PROPERTY ModuleSide : Tc3_Xts_Utility.ModuleSide
GET
ModuleSide := _ModuleSide;
END_GET
SET
_ModuleSide := ModuleSide;
END_SET
END_PROPERTY

PROPERTY Offset : ST_OriginTransform
GET
Offset := _Offset;
END_GET
SET
_Offset := Offset;
END_SET
END_PROPERTY

PROPERTY OTCID : OTCID
GET
OTCID := _Otcid;
END_GET
SET
_Otcid := OTCID;
END_SET
END_PROPERTY

END_FUNCTION_BLOCK

// _Internal/Parts/Tasks/InitializeXtsPartTask
{attribute 'no_explicit_call' := 'This FB is a CLASS and must be accessed using methods or properties'}
FUNCTION_BLOCK InitializeXtsPartTask EXTENDS BaseTaskResult IMPLEMENTS I_XtsPartInitializeTask
VAR
	_Initialized : BOOL;
	_PartId		 : I_XtsPartId;
	_PartUtility : I_ContainXtsPartUtility;
	_Parent		 : I_ContainComponents;
	_Properties	 : I_ContainXtsPartProperties;

	//
	_XtsModuleCollection : I_ContainXtsModules;

	//
	_SubState : UDINT;
END_VAR

METHOD Initialize
VAR
	Module : I_XtsModule;
	pModule	 : POINTER TO XtsModule;
END_VAR
CASE _SubState OF
	0:
		IF _Initialized THEN
			RETURN;
		END_IF

		_Busy	  := TRUE;
		_Error	  := FALSE;
		_ErrorId  := 0;
		_SubState := 10;

	10:
		IF _PartUtility.Utility.GetModuleOids() THEN
			IF _PartUtility.Utility.P_ModuleCount < 1 THEN
				_SubState := 100;
			END_IF

			_XtsModuleCollection.XtsModules.Create(UDINT_TO_UINT(_PartUtility.Utility.P_ModuleCount));
			_SubState := 20;
		END_IF

	20:
		_XtsModuleCollection.XtsModules.ResetIterator();
		WHILE _XtsModuleCollection.XtsModules.MoveToNext DO
			Module := _XtsModuleCollection.XtsModules.Current;
			Module.RegisterWithParent(_Parent);
			Module.Id	   := _XtsModuleCollection.XtsModules.CurrentItem;
			Module.Otcid   := _PartUtility.Utility.P_ModuleOids[_XtsModuleCollection.XtsModules.CurrentItem];
			Module.Utility := _PartUtility.Utility.ModuleTcIo(UDINT_TO_UINT(_XtsModuleCollection.XtsModules.CurrentItem));
		END_WHILE

		_SubState := 30;

	30:
		_Properties.Properties.General.ModuleSide := _PartUtility.Utility.GetModuleSide();
		_Properties.Properties.General.Offset	  := _PartUtility.Utility.GetOriginTransform();
		_Properties.Properties.General.OTCID	  := _PartUtility.Utility.GetTaskOid();
		_SubState								  := 100;

	100:
		_Initialized := TRUE;
		_Busy		 := FALSE;
		_SubState	 := 0;
END_CASE
END_METHOD

{attribute 'monitoring':='call'}
PROPERTY Initialized : BOOL
GET
Initialized := _Initialized;
END_GET
SET
_Initialized := Initialized;
END_SET
END_PROPERTY

PROPERTY XtsPartId : I_XtsPartId
GET
END_GET
SET
_PartId := XtsPartId;
__QUERYINTERFACE(_PartId, _PartUtility);
__QUERYINTERFACE(_PartId, _XtsModuleCollection);
__QUERYINTERFACE(_PartId, _Parent);
__QUERYINTERFACE(_PartId, _Properties);
END_SET
END_PROPERTY

END_FUNCTION_BLOCK

// _Internal/TaskBase/BaseTaskResult
{attribute 'hide_all_locals'}
FUNCTION_BLOCK BaseTaskResult IMPLEMENTS I_TaskResult
VAR
	_TaskName : T_MaxString;
	_Busy	 : BOOL;
	_Error	 : BOOL;
	_ErrorId : UDINT;
END_VAR

{attribute 'monitoring' := 'call'}
PROPERTY Busy : BOOL
GET
Busy := _Busy;
END_GET
END_PROPERTY

{attribute 'monitoring' := 'call'}
PROPERTY Error : BOOL
GET
Error := _Error;
END_GET
END_PROPERTY

{attribute 'monitoring' := 'call'}
PROPERTY ErrorId : UDINT
GET
ErrorId := _ErrorId;
END_GET
END_PROPERTY

{attribute 'monitoring':='call'}
PROPERTY TaskName : STRING
GET
TaskName := _TaskName;
END_GET
SET
_TaskName := TaskName;
END_SET
END_PROPERTY

END_FUNCTION_BLOCK

// _Internal/Parts/Tasks/Interfaces/I_XtsPartInitializeTask
INTERFACE I_XtsPartInitializeTask EXTENDS I_XtsPartTask, I_Initializable

END_INTERFACE

// _Internal/Parts/Tasks/Interfaces/I_XtsPartTask
INTERFACE I_XtsPartTask EXTENDS I_XtsPartTaskResult

PROPERTY XtsPartId : I_XtsPartId
GET
END_GET
SET
END_SET
END_PROPERTY

END_INTERFACE

// _Internal/Parts/Tasks/Interfaces/I_XtsPartTaskResult
INTERFACE I_XtsPartTaskResult EXTENDS I_TaskResult

END_INTERFACE

// _Internal/Collections/Modules/ModuleCollection/XtsModuleCollection
{attribute 'no_explicit_call' := 'This FB is a CLASS and must be accessed using methods or properties'}
{attribute 'enable_dynamic_creation'}
FUNCTION_BLOCK XtsModuleCollection IMPLEMENTS I_XtsModuleCollection, I_Peekable
VAR
	pModuleBuffer	 : POINTER TO PVOID;
	_NumberOfModules : UINT;
	_CurrentModule : I_XtsModule;
	_CurrentIndex  : UDINT := 0;
	{attribute 'hide'}
	_CollectionAdapter : XtsModuleCollectionAdapter(THIS^);
END_VAR

METHOD Clear
VAR
	i	   : UDINT;
	Module : POINTER TO XtsModule;
END_VAR
IF IsEmpty THEN
	RETURN;
END_IF

FOR i := 1 TO _NumberOfModules DO
	Module := GetModuleInstance(i);
	IF Module <> ADR(NullObjects.XtsModule) THEN
		__DELETE(Module);
	END_IF
END_FOR

__DELETE(pModuleBuffer);
_NumberOfModules := 0;
END_METHOD

{attribute 'monitoring' := 'call'}
PROPERTY Count : UDINT
GET
Count := _NumberOfModules;
END_GET
END_PROPERTY

{attribute 'hide'}
METHOD Create : BOOL
VAR_INPUT
	NumberOfModules : UINT;
END_VAR

VAR
	i		 : UINT;
	pModule	 : POINTER TO XtsModule;
	ppBuffer : POINTER TO POINTER TO XtsModule;
END_VAR
IF NOT IsEmpty THEN
	Clear();
END_IF

_NumberOfModules := NumberOfModules;
pModuleBuffer	 := __NEW(PVOID, NumberOfModules);
IF pModuleBuffer <> 0 THEN
	FOR i := 1 TO _NumberOfModules DO
		pModule	  := __NEW(XtsModule(Name := CONCAT('Module ',UINT_TO_STRING(i))));
		ppBuffer  := pModuleBuffer + ((i - 1) * SIZEOF(PVOID));
		ppBuffer^ := pModule;
	END_FOR

	Create := TRUE;
END_IF
END_METHOD

METHOD GetById : I_XtsModule
VAR_INPUT
	ModuleId	: UDINT;
END_VAR
GetById := GetModuleInstance(ModuleId)^;
END_METHOD

METHOD GetByOtcid : I_XtsModule
VAR_INPUT
	ModuleOtcid	: OTCID;
END_VAR
VAR
	i : UDINT;
	ppModule : POINTER TO POINTER TO XtsModule;
END_VAR
GetByOtcid := NullObjects.XtsModule;
FOR i := 0 TO _NumberOfModules DO
	ppModule := pModuleBuffer + ((i) * SIZEOF(PVOID));
	IF ppModule^^.Otcid = ModuleOtcid THEN
		GetByOtcid := ppModule^^;
		RETURN;
	END_IF
END_FOR
END_METHOD

{attribute 'monitoring' := 'call'}
PROPERTY IsEmpty : BOOL
GET
IsEmpty := _NumberOfModules = 0;
END_GET
END_PROPERTY

{attribute 'monitoring':='call'}
PROPERTY Current : I_XtsModule
GET
IF _CurrentModule = 0 THEN
	Current := NullObjects.XtsModule;
ELSE
	Current := _CurrentModule;
END_IF
END_GET
END_PROPERTY

{attribute 'monitoring' := 'call'}
PROPERTY CurrentItem : UDINT
GET
CurrentItem := _CurrentIndex;
END_GET
END_PROPERTY

PROPERTY MoveToNext : BOOL
GET
MoveToNext := FALSE;
IF _NumberOfModules = 0 THEN
	RETURN;
END_IF

IF _CurrentIndex = _NumberOfModules THEN
	RETURN;
END_IF

_CurrentModule := GetById(_CurrentIndex + 1);
_CurrentIndex  := _CurrentIndex + 1;
MoveToNext	   := TRUE;
END_GET
END_PROPERTY

METHOD ResetIterator
_CurrentModule := NullObjects.XtsModule;
_CurrentIndex  := 0;
END_METHOD

METHOD Dispose
VAR
	pDispose : POINTER TO XtsModuleCollection;
END_VAR
Clear();
pDispose := THIS;
__DELETE(pDispose);
END_METHOD

//FB_Exit must be implemented explicitly. If there is an implementation, then the
//method is called before the controller removes the code of the function block instance
//(implicit call). The return value is not evaluated.
METHOD FB_Exit: BOOL
VAR_INPUT
    bInCopyCode: BOOL;  // TRUE: the exit method is called in order to leave the instance which will be copied afterwards (online change).  
END_VAR
IF bInCopyCode THEN
	RETURN;
END_IF

Clear();
END_METHOD

METHOD AcceptPeeker
VAR_INPUT
	Peeker	: Core.I_Peeker;
END_VAR
Peeker.PeekCollection(_CollectionAdapter);
END_METHOD

METHOD PROTECTED CheckModuleId : BOOL
VAR_INPUT
	ModuleId : UDINT;
END_VAR
CheckModuleId := (ModuleId > 0) AND (ModuleId <= _NumberOfModules) AND (pModuleBuffer <> 0);
END_METHOD

METHOD PROTECTED GetModuleInstance : POINTER TO XtsModule
VAR_INPUT
	ModuleId : UDINT; // 1 based index
END_VAR

VAR
	ppModule : POINTER TO POINTER TO XtsModule;
END_VAR
IF CheckModuleId(ModuleId) THEN
	ppModule := pModuleBuffer + ((ModuleId - 1) * SIZEOF(PVOID));
	GetModuleInstance := ppModule^;
ELSE
	GetModuleInstance := ADR(NullObjects.XtsModule);
END_IF
END_METHOD

END_FUNCTION_BLOCK

// _Internal/Collections/Modules/ModuleCollection/Interfaces/XtsModuleCollectionAdapter
FUNCTION_BLOCK XtsModuleCollectionAdapter IMPLEMENTS I_Collection
VAR
	_ModuleCollection : I_XtsModuleCollection;
END_VAR

METHOD AddItem
VAR_INPUT
	Item	: Core.I_Base;
END_VAR
END_METHOD

METHOD Clear
_ModuleCollection.Clear();
END_METHOD

{attribute 'monitoring' := 'call'}
PROPERTY Count : UDINT
GET
Count := _ModuleCollection.Count;
END_GET
END_PROPERTY

PROPERTY Current : Core.I_Base
GET
Current := _ModuleCollection.Current;
END_GET
END_PROPERTY

{attribute 'monitoring' := 'call'}
PROPERTY CurrentItem : UDINT
GET
CurrentItem := _ModuleCollection.CurrentItem;
END_GET
END_PROPERTY

//FB_Init is always available implicitly and it is used primarily for initialization.
//The return value is not evaluated. For a specific influence, you can also declare the
//methods explicitly and provide additional code there with the standard initialization
//code. You can evaluate the return value.
METHOD FB_Init: BOOL
VAR_INPUT
    bInitRetains: BOOL; // TRUE: the retain variables are initialized (reset warm / reset cold)
    bInCopyCode: BOOL;  // TRUE: the instance will be copied to the copy code afterward (online change)
	XtsModuleCollection : I_XtsModuleCollection;   
END_VAR
_ModuleCollection := XtsModuleCollection;
END_METHOD

{attribute 'monitoring' := 'call'}
PROPERTY IsEmpty : BOOL
GET
IsEmpty := _ModuleCollection.IsEmpty;
END_GET
END_PROPERTY

PROPERTY MoveToNext : BOOL
GET
MoveToNext := _ModuleCollection.MoveToNext;
END_GET
END_PROPERTY

METHOD RemoveItem
VAR_INPUT
	Item	: Core.I_Base;
END_VAR
END_METHOD

METHOD ResetIterator
_ModuleCollection.ResetIterator();
END_METHOD

END_FUNCTION_BLOCK

// _Internal/XtsSystem/Properties/Interfaces/I_ContainXtsSystemProperties
INTERFACE I_ContainXtsSystemProperties EXTENDS I_Base

PROPERTY UtilityProperties : I_XtsSystemUtilityProperties
GET
END_GET
END_PROPERTY

END_INTERFACE

// _Internal/XtsSystem/Properties/Interfaces/I_XtsSystemUtilityProperties
INTERFACE I_XtsSystemUtilityProperties EXTENDS I_Base

PROPERTY Mover : I_XtsSystemUtilityPropertiesMover
GET
END_GET
END_PROPERTY

END_INTERFACE

// _Internal/XtsSystem/Properties/Interfaces/I_XtsSystemUtilityPropertiesMover
INTERFACE I_XtsSystemUtilityPropertiesMover EXTENDS I_Base

PROPERTY XtsMagnetPlateType : MagnetPlateType
GET
END_GET
SET
END_SET
END_PROPERTY

PROPERTY XtsMoverType : MoverType
GET
END_GET
SET
END_SET
END_PROPERTY

END_INTERFACE

// _Internal/XtsSystem/Status/Interfaces/I_ContainXtsSystemStatus
INTERFACE I_ContainXtsSystemStatus EXTENDS I_Base

{attribute 'monitoring':='call'}
PROPERTY Status : I_XtsSystemStatus
GET
END_GET
END_PROPERTY

END_INTERFACE

// _Internal/XtsSystem/Status/Interfaces/I_XtsSystemStatus
INTERFACE I_XtsSystemStatus EXTENDS I_Base, I_Cyclic

{attribute 'monitoring':='call'}
PROPERTY NumberOfMovers : UDINT
GET
END_GET
END_PROPERTY

{attribute 'monitoring':='call'}
PROPERTY NumberOfParts : UDINT
GET
END_GET
END_PROPERTY

{attribute 'monitoring':='call'}
PROPERTY NumberOfPositionTriggers : UDINT
GET
END_GET
END_PROPERTY

{attribute 'monitoring':='call'}
PROPERTY NumberOfStations : UDINT
GET
END_GET
END_PROPERTY

{attribute 'monitoring':='call'}
PROPERTY NumberOfTracks : UDINT
GET
END_GET
END_PROPERTY

{attribute 'monitoring':='call'}
PROPERTY NumberOfZones : UDINT
GET
END_GET
END_PROPERTY

{attribute 'monitoring':='call'}
PROPERTY NumberPartsNotReady : USINT
GET
END_GET
END_PROPERTY

{attribute 'monitoring':='call'}
PROPERTY NumberPartsReady : USINT
GET
END_GET
END_PROPERTY

{attribute 'monitoring':='call'}
PROPERTY Simulated : BOOL
GET
END_GET
END_PROPERTY

{attribute 'monitoring':='call'}
PROPERTY Vdc24Okay : BOOL
GET
END_GET
END_PROPERTY

{attribute 'monitoring':='call'}
PROPERTY Vdc48Okay : BOOL
GET
END_GET
END_PROPERTY

END_INTERFACE

// XtsSystem/Interfaces/I_XtsSystemConfiguration
INTERFACE I_XtsSystemConfiguration EXTENDS I_Base

{attribute 'monitoring':='call'}
PROPERTY CommandPositionTriggersOnDisable : BOOL
GET
END_GET
SET
END_SET
END_PROPERTY

{attribute 'monitoring':='call'}
PROPERTY CommandPositionTriggersOnEnable : BOOL
GET
END_GET
SET
END_SET
END_PROPERTY

{attribute 'monitoring':='call'}
PROPERTY CommandStationsOnDisable : BOOL
GET
END_GET
SET
END_SET
END_PROPERTY

{attribute 'monitoring':='call'}
PROPERTY CommandStationsOnEnable : BOOL
GET
END_GET
SET
END_SET
END_PROPERTY

END_INTERFACE

// _Internal/XtsSystem/Base/Interfaces/I_XtsTask
INTERFACE I_XtsTask EXTENDS I_XtsTaskResult

{attribute 'monitoring' := 'call'}
PROPERTY XpuId : I_XtsXpuId
GET
END_GET
SET
END_SET
END_PROPERTY

END_INTERFACE

// _Internal/XtsSystem/Base/Interfaces/I_XtsTaskResult
INTERFACE I_XtsTaskResult EXTENDS I_TaskResult

{attribute 'monitoring':='call'}
PROPERTY TaskId : XtsSystemTaskId
GET
END_GET
END_PROPERTY

END_INTERFACE

// _Internal/XtsSystem/ManualDebugger
FUNCTION_BLOCK ManualDebugger
VAR
	//Xts System Movers Collection
	Movers : CollectionPeeker<5>;
	//Xts System Stations Collection
	Stations : CollectionPeeker<5>;
	//Xts System PositionTriggers Collection
	PositionTriggers : CollectionPeeker<5>;
	//Xts System Zones Collection
	Zones : CollectionPeeker<5>;
	//Xts System XtsParts Collection
	Parts : CollectionPeeker<5>;
	{attribute 'hide'}
	_PartCollection : I_XtsPartCollection;
	//Part defined by PartIdForModules XtsModule Collection
	Modules : CollectionPeeker<5>;
	{attribute 'hide'}
	_PartId			: UDINT := 1;
END_VAR

{attribute 'monitoring':='call'}
PROPERTY PartIdForModules : UDINT
GET
PartIdForModules := _PartId;
END_GET
SET
VAR
	ModulePeekable : I_Peekable;
END_VAR
_PartId := PartIdForModules;

IF __QUERYINTERFACE(_PartCollection.GetById(_PartId).XtsModules, ModulePeekable) THEN
	Modules.CollectionName := CONCAT('Part ', CONCAT(TO_STRING(_PartId), ' Modules'));
	Modules.PeekAt(ModulePeekable);
END_IF
END_SET
END_PROPERTY

PROPERTY RefreshCollections : BOOL
SET
IF NOT RefreshCollections THEN
	RETURN;
END_IF

Movers.Refresh			  := TRUE;
Stations.Refresh		  := TRUE;
PositionTriggers.Refresh := TRUE;
Zones.Refresh			  := TRUE;
Parts.Refresh			  := TRUE;
Modules.Refresh		  := TRUE;
END_SET
END_PROPERTY

METHOD SetCollections
VAR_INPUT
	Movers			 : I_XtsMoverCollection;
	PositionTriggers : I_XtsPositionTriggerCollection;
	Stations		 : I_XtsStationCollection;
	Zones			 : I_XtsZoneCollection;
	Parts			 : I_XtsPartCollection;
END_VAR

VAR
	MoverPeekable	   : I_Peekable;
	PosTriggerPeekable : I_Peekable;
	StationPeekable	   : I_Peekable;
	ZonePeekable	   : I_Peekable;
	PartPeekable	   : I_Peekable;
	ModulePeekable	   : I_Peekable;
END_VAR
IF __QUERYINTERFACE(Movers, MoverPeekable) THEN
	THIS^.Movers.CollectionName := 'Xts System Movers';
	THIS^.Movers.PeekAt(MoverPeekable);
END_IF

IF __QUERYINTERFACE(PositionTriggers, PosTriggerPeekable) THEN
	THIS^.PositionTriggers.CollectionName := 'Xts System Position Triggers';
	THIS^.PositionTriggers.PeekAt(PosTriggerPeekable);
END_IF

IF __QUERYINTERFACE(Stations, StationPeekable) THEN
	THIS^.Stations.CollectionName := 'Xts System Stations';
	THIS^.Stations.PeekAt(StationPeekable);
END_IF

IF __QUERYINTERFACE(Zones, ZonePeekable) THEN
	THIS^.Zones.CollectionName := 'Xts System Zones';
	THIS^.Zones.PeekAt(ZonePeekable);
END_IF

IF __QUERYINTERFACE(Parts, PartPeekable) THEN
	_PartCollection		  := Parts;
	THIS^.Parts.CollectionName := 'Xts System Parts';
	THIS^.Parts.PeekAt(PartPeekable);
END_IF

// IF __QUERYINTERFACE(_PartCollection.GetById(_PartId).XtsModules, ModulePeekable) THEN
// 	THIS^.Modules.CollectionName := CONCAT('Part ', CONCAT(TO_STRING(_PartId), ' Modules'));
// 	THIS^.Modules.PeekAt(ModulePeekable);
// END_IF
END_METHOD

END_FUNCTION_BLOCK

// _Internal/XtsSystem/Base/Interfaces/I_XtsTaskCollection
INTERFACE I_XtsTaskCollection EXTENDS I_Base, I_Cyclic

METHOD AddTask : BOOL
VAR_INPUT
	Task : I_XtsTask;
END_VAR
END_METHOD

METHOD GetTaskById : I_XtsTask
VAR_INPUT
	TaskId : XtsSystemTaskId;
END_VAR
END_METHOD

METHOD GetTaskByName : I_XtsTask
VAR_INPUT
	Name : T_MaxString;
END_VAR
END_METHOD

METHOD RemoveTaskById
VAR_INPUT
	TaskId : XtsSystemTaskId;
END_VAR
END_METHOD

METHOD RemoveTaskByInstance
VAR_INPUT
	Task : I_XtsTask;
END_VAR
END_METHOD

END_INTERFACE

// _Internal/Collections/Movers/MoverCollection/XtsMoverCollection
{attribute 'no_explicit_call' := 'This FB is a CLASS and must be accessed using methods or properties'}
FUNCTION_BLOCK XtsMoverCollection IMPLEMENTS I_XtsMoverCollection, I_Peekable
VAR
	_Collection : Collection<XtsCoreParameters.MaxNumberOfMovers>;
END_VAR

{attribute 'monitoring':='call'}
PROPERTY Current : I_XtsMover
GET
VAR
	Mover : I_XtsMover;
END_VAR
__QUERYINTERFACE(_Collection.Current,Mover);
Current := Mover;
END_GET
END_PROPERTY

{attribute 'monitoring' := 'call'}
PROPERTY CurrentItem : UDINT
GET
CurrentItem := _Collection.CurrentItem;
END_GET
END_PROPERTY

PROPERTY MoveToNext : BOOL
GET
MoveToNext := _Collection.MoveToNext;
END_GET
END_PROPERTY

METHOD ResetIterator
_Collection.ResetIterator();
END_METHOD

METHOD AcceptMoverVisitor
VAR_INPUT
	MoverVisitor : I_XtsMoverVisitor;
END_VAR
VAR
	Mover : I_XtsMover;
END_VAR
_Collection.ResetIterator();
WHILE _Collection.MoveToNext DO
	__QUERYINTERFACE(_Collection.Current, Mover);
	Mover.AcceptMoverVisitor(MoverVisitor);
END_WHILE
END_METHOD

METHOD AcceptPeeker
VAR_INPUT
	Peeker	: Core.I_Peeker;
END_VAR
Peeker.PeekCollection(_Collection);
END_METHOD

METHOD AddItem
VAR_INPUT
	Mover : I_XtsMover;
END_VAR
_Collection.AddItem(Mover);
END_METHOD

METHOD Clear
VAR_INPUT
END_VAR
_Collection.Clear();
END_METHOD

{attribute 'monitoring' := 'call'}
PROPERTY Count : UDINT
GET
Count := _Collection.Count;
END_GET
END_PROPERTY

{attribute 'monitoring':='call'}
PROPERTY IsEmpty : BOOL
GET
IsEmpty := _Collection.IsEmpty;
END_GET
END_PROPERTY

METHOD Map
VAR_INPUT
	Validator : I_XtsMoverValidator;
	Visitor	  : I_XtsMoverVisitor;
END_VAR
VAR
	Mover : I_XtsMover;
END_VAR
_Collection.ResetIterator();
WHILE _Collection.MoveToNext DO
	__QUERYINTERFACE(_Collection.Current, Mover);
	IF Validator.Valid(Mover) THEN
		Visitor.VisitMover(Mover);
	END_IF
END_WHILE
END_METHOD

METHOD Remove
VAR_INPUT
	Mover : I_XtsMover;
END_VAR
_Collection.RemoveItem(Mover);
END_METHOD

END_FUNCTION_BLOCK

// _Internal/Collections/Stations/StationCollection/XtsStationCollection
{attribute 'no_explicit_call' := 'This FB is a CLASS and must be accessed using methods or properties'}
FUNCTION_BLOCK XtsStationCollection IMPLEMENTS I_XtsStationCollection, I_Peekable
VAR
	_Stations : Collection<XtsCoreParameters.MaxNumberOfStations>;
END_VAR

{attribute 'monitoring':='call'}
PROPERTY Current : I_XtsStation
GET
VAR
	Station : I_XtsStation;
END_VAR
__QUERYINTERFACE(_Stations.Current,Station);
Current := Station;
END_GET
END_PROPERTY

{attribute 'monitoring' := 'call'}
PROPERTY CurrentItem : UDINT
GET
CurrentItem := _Stations.CurrentItem;
END_GET
END_PROPERTY

PROPERTY MoveToNext : BOOL
GET
MoveToNext := _Stations.MoveToNext;
END_GET
END_PROPERTY

METHOD ResetIterator
_Stations.ResetIterator();
END_METHOD

METHOD AcceptPeeker
VAR_INPUT
	Peeker	: Core.I_Peeker;
END_VAR
Peeker.PeekCollection(_Stations);
END_METHOD

METHOD AcceptStationVisitor
VAR_INPUT
	StationVisitor : I_XtsStationVisitor;
END_VAR

VAR
	_Station : I_XtsStation;
END_VAR
_Stations.ResetIterator();
WHILE _Stations.MoveToNext DO
	__QUERYINTERFACE(_Stations.Current, _Station);
	_Station.AcceptStationVisitor(StationVisitor);
END_WHILE
END_METHOD

METHOD AddItem
VAR_INPUT
	Station : I_XtsStation;
END_VAR
_Stations.AddItem(Station);
END_METHOD

METHOD Clear
VAR_INPUT
END_VAR
_Stations.Clear();
END_METHOD

{attribute 'monitoring' := 'call'}
PROPERTY Count : UDINT
GET
Count := _Stations.Count;
END_GET
END_PROPERTY

{attribute 'monitoring':='call'}
PROPERTY IsEmpty : BOOL
GET
IsEmpty := _Stations.IsEmpty;
END_GET
END_PROPERTY

METHOD Remove
VAR_INPUT
	Station : I_XtsStation;
END_VAR
_Stations.RemoveItem(Station);
END_METHOD

END_FUNCTION_BLOCK

// _Internal/Collections/PositionTriggers/PositionTriggerCollection/XtsPositionTriggerCollection
{attribute 'no_explicit_call' := 'This FB is a CLASS and must be accessed using methods or properties'}
FUNCTION_BLOCK XtsPositionTriggerCollection IMPLEMENTS I_XtsPositionTriggerCollection, I_Peekable
VAR
	_Collection : Collection<XtsCoreParameters.MaxNumberOfPositionTriggers>;
END_VAR

{attribute 'monitoring':='call'}
PROPERTY Current : I_XtsPositionTrigger
GET
__QUERYINTERFACE(_Collection.Current,Current);
END_GET
END_PROPERTY

{attribute 'monitoring' := 'call'}
PROPERTY CurrentItem : UDINT
GET
CurrentItem := _Collection.CurrentItem;
END_GET
END_PROPERTY

PROPERTY MoveToNext : BOOL
GET
MoveToNext := _Collection.MoveToNext;
END_GET
END_PROPERTY

METHOD ResetIterator
_Collection.ResetIterator();
END_METHOD

METHOD AcceptPeeker
VAR_INPUT
	Peeker	: Core.I_Peeker;
END_VAR
Peeker.PeekCollection(_Collection);
END_METHOD

METHOD AcceptXtsPositionTriggerVisitor
VAR_INPUT
	PositionTriggerVisitor : I_VisitXtsPositionTrigger;
END_VAR

VAR
	_PositionTrigger : I_XtsPositionTrigger;
END_VAR
_Collection.ResetIterator();
WHILE _Collection.MoveToNext DO
	__QUERYINTERFACE(_Collection.Current, _PositionTrigger);
	PositionTriggerVisitor.VisitXtsPositionTrigger(_PositionTrigger);
END_WHILE
END_METHOD

METHOD AddItem
VAR_INPUT
	PositionTrigger : I_XtsPositionTrigger;
END_VAR
_Collection.AddItem(PositionTrigger);
END_METHOD

METHOD Clear
VAR_INPUT
END_VAR
_Collection.Clear();
END_METHOD

{attribute 'monitoring' := 'call'}
PROPERTY Count : UDINT
GET
Count := _Collection.Count;
END_GET
END_PROPERTY

{attribute 'monitoring':='call'}
PROPERTY IsEmpty : BOOL
GET
IsEmpty := _Collection.IsEmpty;
END_GET
END_PROPERTY

METHOD Remove
VAR_INPUT
	PositionTrigger : I_XtsPositionTrigger;
END_VAR
_Collection.RemoveItem(PositionTrigger);
END_METHOD

END_FUNCTION_BLOCK

// _Internal/Collections/Zones/ZoneCollection/XtsZoneCollection
{attribute 'no_explicit_call' := 'This FB is a CLASS and must be accessed using methods or properties'}
FUNCTION_BLOCK XtsZoneCollection IMPLEMENTS I_XtsZoneCollection, I_Peekable
VAR
	_Zones : Collection<XtsCoreParameters.MaxNumberOfZones>;
END_VAR

{attribute 'monitoring':='call'}
PROPERTY Current : I_XtsZone
GET
VAR
	Zone : I_XtsZone;
END_VAR
__QUERYINTERFACE(_Zones.Current,Zone);
Current := Zone;
END_GET
END_PROPERTY

{attribute 'monitoring' := 'call'}
PROPERTY CurrentItem : UDINT
GET
CurrentItem := _Zones.CurrentItem;
END_GET
END_PROPERTY

PROPERTY MoveToNext : BOOL
GET
MoveToNext := _Zones.MoveToNext;
END_GET
END_PROPERTY

METHOD ResetIterator
_Zones.ResetIterator();
END_METHOD

METHOD AcceptPeeker
VAR_INPUT
	Peeker	: Core.I_Peeker;
END_VAR
Peeker.PeekCollection(_Zones);
END_METHOD

METHOD AddItem
VAR_INPUT
	Zone : I_XtsZone;
END_VAR
_Zones.AddItem(Zone);
END_METHOD

METHOD Clear
VAR_INPUT
END_VAR
_Zones.Clear();
END_METHOD

{attribute 'monitoring' := 'call'}
PROPERTY Count : UDINT
GET
Count := _Zones.Count;
END_GET
END_PROPERTY

{attribute 'monitoring':='call'}
PROPERTY IsEmpty : BOOL
GET
IsEmpty := _Zones.IsEmpty;
END_GET
END_PROPERTY

METHOD Remove
VAR_INPUT
	Zone : I_XtsZone;
END_VAR
_Zones.RemoveItem(Zone);
END_METHOD

END_FUNCTION_BLOCK

// XtsSystem/XtsSystem
{attribute 'no_explicit_call' := 'This FB is a CLASS and must be accessed using methods or properties'}
FUNCTION_BLOCK XtsSystem EXTENDS Module IMPLEMENTS I_XtsSystem
VAR
	_DefaultTaskCollection : XtsTaskCollection<10>(THIS^);
	_TaskCollection		   : I_XtsTaskCollection := _DefaultTaskCollection;
	_Tasks				   : _XtsTasks;
	_CurrentTask		   : I_XtsTask := NullObjects.XtsTask;
	_XpuId				   : USINT;
	{attribute 'hide'}
	_Error : BOOL;
	{attribute 'hide'}
	_Busy : BOOL;
	{attribute 'hide'}
	_ErrorId : UDINT;

	//
	{attribute 'hide'}
	_Config		  : XtsSystemConfiguration;
	_AxesGroupRef : AXES_GROUP_REF;
	{attribute 'hide'}
	_MoverCommander : XtsMoverCommander;
	_GroupController : XtsGroupController('XtsSystem CA Group Controller');
	{attribute 'hide'}
	_MoverCollection : XtsMoverCollection;
	{attribute 'hide'}
	_DefaultPartCollection : XtsPartCollection;
	{attribute 'hide'}
	_PartCollection : I_XtsPartCollection := _DefaultPartCollection;
	{attribute 'hide'}
	_Status : XtsSystemStatus(THIS^);
	{attribute 'hide'}
	_StationCollection : XtsStationCollection;
	{attribute 'hide'}
	_PositionTriggerCollection : XtsPositionTriggerCollection;
	{attribute 'hide'}
	_ZoneCollection : XtsZoneCollection;
	{attribute 'hide'}
	_DefaultTrackCollection : XtsTrackCollection;
	{attribute 'hide'}
	_TrackCollection : I_XtsTrackCollection := _DefaultTrackCollection;
	{attribute 'hide'}
	_Environment : I_TcIoXtsEnvironment;
	{attribute 'hide'}
	_XpuUtility : I_TcIoXtsProcessingUnit;
	{attribute 'hide'}
	_LocalLogger : XtsLocalLogger;
	{attribute 'hide'}
	_Logger			   : XtsTracePublisher;
	_UtilityProperties : XtsSystemUtilityProperties;
	_MainTrack		   : XtsTrack;
	_Enabled		   : BOOL;
	enableState		   : UDINT;
	{attribute 'hide'}
	_ManualDebugger : ManualDebugger;
END_VAR

{attribute 'monitoring':='call'}
PROPERTY Movers : I_XtsMoverCollection
GET
Movers := _MoverCollection;
END_GET
END_PROPERTY

{attribute 'monitoring' := 'call'}
PROPERTY Parameters : I_XtsParameterSet
GET
Parameters := _MoverCommander.Parameters;
END_GET
SET
_MoverCommander.Parameters.CopyFrom(Parameters);
END_SET
END_PROPERTY

PROPERTY Parts : I_XtsPartCollection
GET
Parts := _PartCollection;
END_GET
END_PROPERTY

PROPERTY PositionTriggers : I_XtsPositionTriggerCollection
GET
PositionTriggers := _PositionTriggerCollection;
END_GET
END_PROPERTY

PROPERTY Stations : I_XtsStationCollection
GET
Stations := _StationCollection;
END_GET
END_PROPERTY

PROPERTY Tracks : I_XtsTrackCollection
GET
Tracks := _TrackCollection;
END_GET
END_PROPERTY

PROPERTY XtsTasks : I_XtsTaskCollection
GET
XtsTasks := _TaskCollection;
END_GET
END_PROPERTY

PROPERTY Zones : I_XtsZoneCollection
GET
Zones := _ZoneCollection;
END_GET
END_PROPERTY

METHOD Disable
_Tasks.DisableXtsTask.Execute();
_CurrentTask := _Tasks.DisableXtsTask;
END_METHOD

METHOD DisableGroup
VAR_INPUT
END_VAR
_GroupController.Disable();
END_METHOD

METHOD DisableMovers
VAR_INPUT
END_VAR
VAR
	Mover : I_XtsMover;
END_VAR
_MoverCollection.ResetIterator();
WHILE _MoverCollection.MoveToNext DO
	Mover := _MoverCollection.Current;
	IF Mover.Enabled THEN
		Mover.Disable();
	END_IF
END_WHILE
END_METHOD

METHOD Enable
_Tasks.EnableXtsTask.Execute();
_CurrentTask := _Tasks.EnableXtsTask;
END_METHOD

METHOD EnableGroup
VAR_INPUT
END_VAR
_GroupController.Enable();
END_METHOD

METHOD EnableMovers
VAR_INPUT
END_VAR
VAR
	Mover : I_XtsMover;
END_VAR
_MoverCollection.ResetIterator();
WHILE _MoverCollection.MoveToNext DO
	Mover := _MoverCollection.Current;
	IF NOT Mover.Enabled THEN
		Mover.Enable();
	END_IF
END_WHILE
END_METHOD

METHOD Reset
_DefaultTaskCollection.Reset();
_GroupController.Reset();
_MoverCollection.ResetIterator();
WHILE _MoverCollection.MoveToNext DO
	IF _MoverCollection.Current.Error THEN
		_MoverCollection.Current.Reset();	
	END_IF
END_WHILE

_Busy	 := FALSE;
_Error	 := FALSE;
_ErrorId := 0;
END_METHOD

METHOD ResetCaGroup
VAR_INPUT
END_VAR
_GroupController.Reset();
END_METHOD

METHOD ResetMovers
VAR_INPUT
END_VAR
_MoverCollection.ResetIterator();
WHILE _MoverCollection.MoveToNext DO
	IF _MoverCollection.Current.Error THEN
		_MoverCollection.Current.Reset();	
	END_IF
END_WHILE
END_METHOD

METHOD RetriggerMoverDetection
VAR_INPUT
END_VAR
_Tasks.MoverRedetectionTask.Execute();
_CurrentTask := _Tasks.MoverRedetectionTask;
END_METHOD

METHOD TriggerMoverDetection
VAR_INPUT
END_VAR
_Tasks.MoverDetectionTask.Execute();
_CurrentTask := _Tasks.MoverDetectionTask;
END_METHOD

METHOD TriggerMoverIdentification
VAR_INPUT
END_VAR
_Tasks.MoverIdentificationTask.Execute();
_CurrentTask := _Tasks.MoverIdentificationTask;
END_METHOD

//FB_Init is always available implicitly and it is used primarily for initialization.

//The return value is not evaluated. For a specific influence, you can also declare the

//methods explicitly and provide additional code there with the standard initialization

//code. You can evaluate the return value.
METHOD FB_Init : BOOL
VAR_INPUT
	bInitRetains		: BOOL;				 // TRUE: the retain variables are initialized (reset warm / reset cold)
	bInCopyCode			: BOOL;				 // TRUE: the instance will be copied to the copy code afterward (online change)  
	Name				: T_MaxString;		 //Name of the XPU the system will interface with
END_VAR
CyclicRunner.AddCallee(_Status);
_GroupController.RegisterWithParent(THIS^);
_GroupController.AxesGroup REF= _AxesGroupRef;
_Logger.Subscribe(_LocalLogger);
IF XtsCoreParameters.TcEventLoggerEnabled THEN
	_Logger.Subscribe(XtsTrace.EventLogger);
END_IF

_ManualDebugger.SetCollections(_MoverCollection,
							   _PositionTriggerCollection,
							   _StationCollection,
							   _ZoneCollection,
							   _PartCollection);

_Tasks.EnableXtsTask.XtsMoverCommander		  := _MoverCommander;
_Tasks.EnableXtsTask.XtsMoverGroupController  := _GroupController;
_Tasks.EnableXtsTask.AxesGroup				  REF= _AxesGroupRef;
_Tasks.DisableXtsTask.XtsMoverCommander		  := _MoverCommander;
_Tasks.DisableXtsTask.XtsMoverGroupController := _GroupController;
_Tasks.DisableXtsTask.AxesGroup				  REF= _AxesGroupRef;
_TaskCollection.AddTask(_Tasks.MoverIdentificationTask);
_TaskCollection.AddTask(_Tasks.MoverDetectionTask);
_TaskCollection.AddTask(_Tasks.MoverRedetectionTask);
_TaskCollection.AddTask(_Tasks.InitializeXtsTask);
_TaskCollection.AddTask(_Tasks.EnableXtsTask);
_TaskCollection.AddTask(_Tasks.DisableXtsTask);
RegisterCyclic(_TaskCollection);
END_METHOD

METHOD Initializing
IF _Tasks.InitializeXtsTask.Initialized THEN //Can only intialize once
	RETURN;
END_IF

_Tasks.InitializeXtsTask.Initialize();
_TaskCollection.CyclicLogic();
ModuleInitialized := _Tasks.InitializeXtsTask.Initialized;
_CurrentTask	  := _Tasks.InitializeXtsTask;
END_METHOD

PROPERTY UtilityProperties : I_XtsSystemUtilityProperties
GET
UtilityProperties := _UtilityProperties;
END_GET
END_PROPERTY

{attribute 'monitoring':='call'}
PROPERTY AxesGroupRef : REFERENCE TO AXES_GROUP_REF
GET
AxesGroupRef REF= _AxesGroupRef;
END_GET
END_PROPERTY

{attribute 'monitoring':='call'}
PROPERTY Busy : BOOL
GET
Busy := _Busy;
END_GET
END_PROPERTY

{attribute 'monitoring' := 'call'}
PROPERTY CAGroupErrorId : UDINT
GET
CAGroupErrorId := _GroupController.ErrorId;
END_GET
END_PROPERTY

{attribute 'monitoring' := 'call'}
PROPERTY CaGroupStatus : E_MoverGroupState
GET
CaGroupStatus := _GroupController.GroupStatus;
END_GET
END_PROPERTY

{attribute 'monitoring':='call'}
PROPERTY Config : I_XtsSystemConfiguration
GET
Config := _Config;
END_GET
END_PROPERTY

{attribute 'monitoring':='call'}
PROPERTY CurrentTask : I_XtsTask
GET
CurrentTask := _CurrentTask;
END_GET
END_PROPERTY

{attribute 'monitoring' := 'call'}
PROPERTY Enabled : BOOL
GET
Enabled := _Enabled; //_XpuUtility.GetDriveState() >= DriveState.SwitchedOn ;
END_GET
END_PROPERTY

PROPERTY Environment : I_TcIoXtsEnvironment
GET
Environment := _Environment;
END_GET
SET
_Environment := Environment;
END_SET
END_PROPERTY

{attribute 'monitoring':='call'}
PROPERTY Error : BOOL
GET
Error := _Error;
END_GET
END_PROPERTY

{attribute 'monitoring':='call'}
PROPERTY ErrorId : UDINT
GET
ErrorId := _ErrorId;
END_GET
END_PROPERTY

{attribute 'monitoring' := 'call'}
PROPERTY MoversEnabled : BOOL
GET
IF _XpuUtility = 0 THEN
	MoversEnabled := FALSE;
	RETURN;
END_IF

MoversEnabled := _XpuUtility.GetDriveState() >= DriveState.SwitchedOn;
END_GET
END_PROPERTY

{attribute 'monitoring':='call'}
PROPERTY Status : I_XtsSystemStatus
GET
Status := _Status;
END_GET
END_PROPERTY

PROPERTY Utility : I_TcIoXtsProcessingUnit
GET
Utility := _XpuUtility;
END_GET
SET
_XpuUtility := Utility;
END_SET
END_PROPERTY

{attribute 'monitoring':='call'}
PROPERTY XpuId : USINT
GET
XpuId := _XpuId;
END_GET
END_PROPERTY

{attribute 'monitoring':='call'}
PROPERTY CommandLog : I_XtsLocalLog
GET
CommandLog := _LocalLogger;
END_GET
END_PROPERTY

PROPERTY TracePublisher : I_XtsTracePublisher
GET
TracePublisher := _Logger;
END_GET
END_PROPERTY

METHOD AcceptMoverVisitor
VAR_INPUT
	MoverVisitor : I_XtsMoverVisitor;
END_VAR
_MoverCollection.AcceptMoverVisitor(MoverVisitor);
END_METHOD

METHOD AcceptStationVisitor
VAR_INPUT
	StationVisitor : I_XtsStationVisitor;
END_VAR
_StationCollection.ResetIterator();
WHILE _StationCollection.MoveToNext DO
	_StationCollection.Current.AcceptStationVisitor(StationVisitor);
END_WHILE
END_METHOD

METHOD AcceptXtsModuleVisitor
VAR_INPUT
	XtsModuleVisitor : I_XtsModuleVisitor;
END_VAR
_PartCollection.ResetIterator();
WHILE _PartCollection.MoveToNext DO
	_PartCollection.Current.AcceptXtsModuleVisitor(XtsModuleVisitor);
END_WHILE
END_METHOD

METHOD AcceptXtsPartVisitor
VAR_INPUT
	XtsPartVisitor : I_XtsPartVisitor;
END_VAR
_PartCollection.ResetIterator();
WHILE _PartCollection.MoveToNext DO
	_PartCollection.Current.AcceptXtsPartVisitor(XtsPartVisitor);
END_WHILE
END_METHOD

METHOD AcceptXtsPositionTriggerVisitor
VAR_INPUT
	PositionTriggerVisitor : I_VisitXtsPositionTrigger;
END_VAR
_PositionTriggerCollection.ResetIterator();
WHILE _PositionTriggerCollection.MoveToNext DO
	_PositionTriggerCollection.Current.AcceptXtsPositionTriggerVisitor(PositionTriggerVisitor);
END_WHILE
END_METHOD

METHOD AcceptXtsZoneVisitor
VAR_INPUT
	ZoneVisitor : I_XtsZoneVisitor;
END_VAR
_ZoneCollection.ResetIterator();
WHILE _ZoneCollection.MoveToNext DO
	_ZoneCollection.Current.AcceptXtsZoneVisitor(ZoneVisitor);
END_WHILE
END_METHOD

{attribute 'monitoring':='call'}
PROPERTY ManualDiagnoser : REFERENCE TO ManualDebugger
GET
ManualDiagnoser REF= _ManualDebugger;
END_GET
END_PROPERTY

METHOD OnCyclicCall
VAR
	InitTask : I_Cyclic;
END_VAR
IF NOT Initialized THEN
	RETURN;
END_IF

//TODO: Improve
CASE enableState OF
	0:
		IF NOT _Enabled AND _Tasks.EnableXtsTask.Busy THEN
			enableState := 1;
		END_IF

	1:
		IF NOT _Tasks.EnableXtsTask.Busy AND NOT _Tasks.EnableXtsTask.Error THEN
			_Enabled	:= TRUE;
			enableState := 2;
		END_IF

	2:
		IF _Tasks.DisableXtsTask.Busy THEN
			enableState := 3;
		END_IF

	3:
		IF NOT _Tasks.DisableXtsTask.Busy AND NOT _Tasks.EnableXtsTask.Error THEN
			_Enabled	:= FALSE;
			enableState := 0;
		END_IF
END_CASE

_Busy	 := _DefaultTaskCollection.Busy;
_Error	 := _DefaultTaskCollection.Error;
_ErrorId := _DefaultTaskCollection.ErrorId;
_MoverCollection.ResetIterator();
WHILE _MoverCollection.MoveToNext DO
	_Busy  := _Busy OR _MoverCollection.Current.Busy;
	_Error := _Error OR _MoverCollection.Current.Error;
	IF _ErrorId = 0 THEN
		_ErrorId := _MoverCollection.Current.ErrorId;
	END_IF
END_WHILE

_Error := _Error OR _GroupController.Error;
END_METHOD

END_FUNCTION_BLOCK

// _Internal/XtsSystem/Base/XtsTaskCollection
{attribute 'no_explicit_call' := 'This FB is a CLASS and must be accessed using methods or properties'}
FUNCTION_BLOCK XtsTaskCollection 
VAR_GENERIC CONSTANT
	MaxCount : UDINT := 10;
END_VAR
IMPLEMENTS I_XtsTaskCollection
VAR
	{attribute 'hide'}
	_NullXtsTask   :  NullXtsTask;
	_XpuId		   : I_XtsXpuId;
	TaskCollection : ARRAY[0..MaxCount - 1] OF I_XtsTask;
	_TaskCount 	   : UDINT;
	_Error : BOOL;
	_Busy : BOOL;
	_ErrorId : UDINT;
END_VAR

METHOD AddTask : BOOL
VAR_INPUT
	Task	: I_XtsTask;
END_VAR
IF _TaskCount = MaxCount THEN
	AddTask := FALSE;
	RETURN;
END_IF

Task.XpuId					:= _XpuId;
TaskCollection[Task.TaskId] := Task;
_TaskCount					:= _TaskCount + 1;
AddTask						:= TRUE;
END_METHOD

{attribute 'monitoring':='call'}
PROPERTY Busy : BOOL
GET
Busy := _Busy;
END_GET
END_PROPERTY

METHOD CyclicLogic
VAR
	Cyclic : I_Cyclic;
	i	   : UDINT;
END_VAR
_Busy := FALSE;
FOR i := 0 TO MaxCount - 1 DO
	IF TaskCollection[i] = 0 THEN
		CONTINUE;
	END_IF
	IF TaskCollection[i].Busy THEN
		_Busy := TRUE;
	END_IF
	IF TaskCollection[i].Error AND NOT _Error THEN
		_Error := TRUE;
		_ErrorId := TaskCollection[i].ErrorId;
	END_IF
	__QUERYINTERFACE(TaskCollection[i], Cyclic);
	IF Cyclic = 0 THEN
		CONTINUE;
	END_IF

	Cyclic.CyclicLogic();
END_FOR
END_METHOD

{attribute 'monitoring':='call'}
PROPERTY Error : BOOL
GET
Error := _Error;
END_GET
END_PROPERTY

{attribute 'monitoring':='call'}
PROPERTY ErrorId : UDINT
GET
ErrorId := _ErrorId;
END_GET
END_PROPERTY

//FB_Init is always available implicitly and it is used primarily for initialization.

//The return value is not evaluated. For a specific influence, you can also declare the

//methods explicitly and provide additional code there with the standard initialization

//code. You can evaluate the return value.
METHOD FB_Init : BOOL
VAR_INPUT
	bInitRetains : BOOL; // TRUE: the retain variables are initialized (reset warm / reset cold)
	bInCopyCode	 : BOOL; // TRUE: the instance will be copied to the copy code afterward (online change)
	XpuId		 : I_XtsXpuId;
END_VAR
VAR
	i : UDINT;
END_VAR
_XpuId := XpuId;
FOR i := 0 TO MaxCount - 1 DO
	TaskCollection[i] := _NullXtsTask;
END_FOR
END_METHOD

METHOD GetTaskById : I_XtsTask
VAR_INPUT
	TaskId : XtsSystemTaskId;
END_VAR
GetTaskById := TaskCollection[TaskId];
END_METHOD

METHOD GetTaskByName : I_XtsTask
VAR_INPUT
	Name : T_MaxString;
END_VAR

VAR
	i : UDINT;
END_VAR
GetTaskByName := _NullXtsTask;
FOR i:=0 TO _TaskCount - 1 DO
	IF TaskCollection[i].TaskName = Name THEN
		GetTaskByName := TaskCollection[i];
		RETURN;
	END_IF
END_FOR
END_METHOD

METHOD RemoveTaskById
VAR_INPUT
	TaskId : XtsSystemTaskId;
END_VAR
TaskCollection[TaskId] := _NullXtsTask;
_TaskCount			   := _TaskCount - 1;
END_METHOD

METHOD RemoveTaskByInstance
VAR_INPUT
	Task	: I_XtsTask;
END_VAR
TaskCollection[Task.TaskId] := _NullXtsTask;
_TaskCount					:= _TaskCount - 1;
END_METHOD

METHOD Reset
VAR_INPUT
END_VAR

VAR
	i		   : UDINT;
	Resettable : I_Resettable;
END_VAR
FOR i := 0 TO MaxCount - 1 DO
	IF TaskCollection[i] = 0 THEN
		CONTINUE;
	END_IF

	IF __QUERYINTERFACE(TaskCollection[i], Resettable) THEN
		Resettable.Reset();
	END_IF
END_FOR

_Busy	 := FALSE;
_Error	 := FALSE;
_ErrorId := 0;
END_METHOD

END_FUNCTION_BLOCK

// _Internal/NullObjects/NullXtsTask
{attribute 'no_explicit_call' := 'This FB is a CLASS and must be accessed using methods or properties'}
{attribute 'conditionalshow'}
{warning disable C0094}
{warning disable C0568}
FUNCTION_BLOCK NullXtsTask IMPLEMENTS I_XtsTask, I_NullObject
VAR
END_VAR

PROPERTY Busy : BOOL
GET
END_GET
END_PROPERTY

PROPERTY Error : BOOL
GET
END_GET
END_PROPERTY

PROPERTY ErrorId : UDINT
GET
END_GET
END_PROPERTY

PROPERTY TaskId : XtsSystemTaskId
GET
END_GET
END_PROPERTY

PROPERTY TaskName : STRING
GET
END_GET
END_PROPERTY

PROPERTY XpuId : I_XtsXpuId
GET
END_GET
SET
END_SET
END_PROPERTY

END_FUNCTION_BLOCK

// _Internal/NullObjects/I_NullObject
INTERFACE I_NullObject EXTENDS I_Base

END_INTERFACE

// _Internal/XtsSystem/Tasks/_XtsTasks
{attribute 'no_explicit_call' := 'This FB is a CLASS and must be accessed using methods or properties'}
FUNCTION_BLOCK _XtsTasks
VAR
	_DefaultTasks			 : _DefaultXtsTasks;
	_EnableXtsTask			 : I_XtsEnableTask				:= _DefaultTasks.EnableXtsTask;
	_InitializeXtsTask		 : I_XtsInitializeTask			:= _DefaultTasks.InitializeXtsTask;
	_DisableXtsTask			 : I_XtsDisableTask				:= _DefaultTasks.DisableXtsTask;
	_MoverDetectionTask		 : I_XtsMoverDetectionTask		:= _DefaultTasks.MoverDetectionTask;
	_MoverRedetectionTask	 : I_XtsMoverRedetectionTask	:= _DefaultTasks.MoverRedetectionTask;
	_MoverIdentificationTask : I_XtsMoverIdentificationTask := _DefaultTasks.MoverIdentificationTask;
END_VAR

{attribute 'monitoring' := 'call'}
PROPERTY DisableXtsTask : I_XtsDisableTask
GET
DisableXtsTask := _DisableXtsTask;
END_GET
SET
_DisableXtsTask := DisableXtsTask;
END_SET
END_PROPERTY

{attribute 'monitoring' := 'call'}
PROPERTY EnableXtsTask : I_XtsEnableTask
GET
EnableXtsTask := _EnableXtsTask;
END_GET
SET
_EnableXtsTask := EnableXtsTask;
END_SET
END_PROPERTY

{attribute 'monitoring' := 'call'}
PROPERTY InitializeXtsTask : I_XtsInitializeTask
GET
InitializeXtsTask := _InitializeXtsTask;
END_GET
SET
_InitializeXtsTask := InitializeXtsTask;
END_SET
END_PROPERTY

{attribute 'monitoring' := 'call'}
PROPERTY MoverDetectionTask : I_XtsMoverDetectionTask
GET
MoverDetectionTask := _MoverDetectionTask;
END_GET
SET
_MoverDetectionTask := MoverDetectionTask;
END_SET
END_PROPERTY

{attribute 'monitoring' := 'call'}
PROPERTY MoverIdentificationTask : I_XtsMoverIdentificationTask
GET
MoverIdentificationTask := _MoverIdentificationTask;
END_GET
SET
_MoverIdentificationTask := MoverIdentificationTask;
END_SET
END_PROPERTY

{attribute 'monitoring' := 'call'}
PROPERTY MoverRedetectionTask : I_XtsMoverRedetectionTask
GET
MoverRedetectionTask  := _MoverRedetectionTask;
END_GET
SET
_MoverRedetectionTask := MoverRedetectionTask;
END_SET
END_PROPERTY

END_FUNCTION_BLOCK

// _Internal/XtsSystem/Tasks/_DefaultXtsTasks
{attribute 'no_explicit_call' := 'This FB is a CLASS and must be accessed using methods or properties'}
FUNCTION_BLOCK _DefaultXtsTasks
VAR
	EnableXtsTask			: EnableXtsTask;
	InitializeXtsTask		: InitializeXtsTask;
	DisableXtsTask			: DisableXtsTask;
	MoverDetectionTask		: MoverDetectionTask;
	MoverRedetectionTask	: MoverRedetectionTask;
	MoverIdentificationTask : MoverIdentificationTask;
END_VAR

END_FUNCTION_BLOCK

// _Internal/XtsSystem/Tasks/EnableXtsTask
{attribute 'no_explicit_call' := 'This FB is a CLASS and must be accessed using methods or properties'}
FUNCTION_BLOCK EnableXtsTask EXTENDS XtsTaskResult IMPLEMENTS I_XtsEnableTask, I_Cyclic
VAR
	_XpuId					   : I_XtsXpuId;
	_XtsSystem				   : I_XtsSystem;
	_XtsStatus				   : I_ContainXtsSystemStatus;
	_State					   : UDINT;
	_MoverCommander			   : I_XtsMoverCommander;
	_GroupController		   : I_XtsMoverGroupController;
	_PositionTriggerCollection : I_XtsPositionTriggerCollection;
	_StationCollection		   : I_XtsStationCollection;
	_ZoneCollection			   : I_XtsZoneCollection;
	_MoverIdTask			   : I_XtsMoverIdentificationTask;
	_AxesGroup				   : REFERENCE TO AXES_GROUP_REF;

	//CA Group Parameters
	_CollisionAvoidanceGroupParameters : I_CollisionAvoidanceGroupable;
	
	//
	WatchdogCheck	 : UDINT;
	ExecuteWatchdog	 : UDINT;
END_VAR

PROPERTY AxesGroup : REFERENCE TO AXES_GROUP_REF
GET
AxesGroup REF= _AxesGroup;
END_GET
SET
_AxesGroup REF= AxesGroup;
END_SET
END_PROPERTY

METHOD CyclicLogic
VAR
	_Check	   : BOOL;
	AxesGroup : REFERENCE TO AXES_GROUP_REF;
	LogSource  : TraceSourceInfo;
	LogMessage : TraceMessageInfo;
END_VAR
LogSource.SourceName := 'EnableXtsTask';
IF ExecuteWatchdog <> WatchdogCheck THEN
	WatchdogCheck := ExecuteWatchdog;
ELSE
	ExecuteWatchdog	 := 0;
	_CommandExecuted := FALSE;
END_IF

CASE _State OF
	0:
		IF _CommandExecuted THEN
			_Busy				 := TRUE;
			_Error				 := FALSE;
			_ErrorId			 := 0;
			LogMessage.Message	 := 'System Enable Started.';
			LogMessage.MessageId := E_XtsLogMessage.SystemInfo;
			LogMessage.Severity	 := 1;
			_Logger.LogMessageInstance(LogSource, LogMessage);
			IF _XtsStatus.Status.Simulated THEN
				LogMessage.Message	 := 'Xts System Simulated. Voltage check skipped.';
				LogMessage.MessageId := E_XtsLogMessage.SystemVerbose;
				LogMessage.Severity	 := 0;
				_Logger.LogMessageInstance(LogSource, LogMessage);
				_State := 11;
			ELSE
				_State := 10;
			END_IF
		END_IF

	10:
		//Check  voltage
		IF _XtsStatus.Status.VDC24Okay AND _XtsStatus.Status.VDC48Okay THEN
			LogMessage.Message	 := 'Xts Voltage check okay.';
			LogMessage.MessageId := E_XtsLogMessage.SystemVerbose;
			LogMessage.Severity	 := 0;
			_Logger.LogMessageInstance(LogSource, LogMessage);
			_State := 11;
		ELSE
			LogMessage.Message	 := 'Xts Voltage not okay! Check 24/48v on modules.';
			LogMessage.MessageId := E_XtsLogMessage.SystemEnableVoltageCheckFailed;
			LogMessage.Severity	 := 3;
			_Logger.LogMessageInstance(LogSource, LogMessage);
			_State := 255;
		END_IF

	11:
		IF _XtsSystem.Utility.GetIsMoverIdDetectionValid() THEN
			LogMessage.Message	 := 'XtsMover Identification Already Valid, skipped.';
			LogMessage.MessageId := E_XtsLogMessage.SystemVerbose;
			LogMessage.Severity	 := 0;
			_Logger.LogMessageInstance(LogSource, LogMessage);
			_State := 20;
		ELSE
			_MoverIdTask.Execute();
			_State := 12;
		END_IF

	12:
		IF _MoverIdTask.Error THEN
			LogMessage.Message	 := CONCAT('Mover Identification failed: ', TO_STRING(_MoverIdTask.ErrorId));
			LogMessage.MessageId := E_XtsLogMessage.SystemError;
			LogMessage.Severity	 := 4;
			_Logger.LogMessageInstance(LogSource, LogMessage);
			_ErrorId := _MoverIdTask.ErrorId;
			_Error	 := TRUE;
			_State	 := 255;
		ELSIF NOT _MoverIdTask.Busy THEN
			LogMessage.Message	 := 'XtsMover Identification finished.';
			LogMessage.MessageId := E_XtsLogMessage.SystemVerbose;
			LogMessage.Severity	 := 0;
			_Logger.LogMessageInstance(LogSource, LogMessage);
			_State := 20;
		END_IF

	20:
		_MoverCommander.Enable(_XtsSystem.Movers);
		_State := 30;

	30:
		//Enable all movers
		IF _MoverCommander.Error THEN
			LogMessage.Message	 := CONCAT('Movers failed to enable: ', TO_STRING(_MoverCommander.ErrorId));
			LogMessage.MessageId := E_XtsLogMessage.SystemError;
			LogMessage.Severity	 := 4;
			_Logger.LogMessageInstance(LogSource, LogMessage);
			_Error := TRUE;
			_State := 255;
		ELSIF NOT _MoverCommander.Busy THEN
			LogMessage.Message	 := 'XtsMovers all movers enabled.';
			LogMessage.MessageId := E_XtsLogMessage.SystemVerbose;
			LogMessage.Severity	 := 0;
			_Logger.LogMessageInstance(LogSource, LogMessage);
			AxesGroup REF= _AxesGroup;
			_MoverCommander.AddToGroup(_XtsSystem.Movers, AxesGroup, 1);
			_State := 40;
		END_IF

	40:
		//Add all to Xts Group
		IF _MoverCommander.Error THEN
			LogMessage.Message	 := CONCAT('Movers failed to Add to CA Group: ', TO_STRING(_MoverCommander.ErrorId));
			LogMessage.MessageId := E_XtsLogMessage.SystemError;
			LogMessage.Severity	 := 4;
			_Logger.LogMessageInstance(LogSource, LogMessage);
			_Error := TRUE;
			_State := 255;
			_Error := TRUE;
			_State := 255;
		ELSIF NOT _MoverCommander.Busy THEN
			_GroupController.Enable();
			_State := 50;
		END_IF

	50:
		//Enable the XTS Group
		IF _GroupController.Error THEN
			LogMessage.Message	 := CONCAT('Failed to Enable CA Group: ', TO_STRING(_GroupController.ErrorId));
			LogMessage.MessageId := E_XtsLogMessage.SystemError;
			LogMessage.Severity	 := 4;
			_Logger.LogMessageInstance(LogSource, LogMessage);
			_Error := TRUE;
			_State := 255;
			_Error := TRUE;
			_State := 255;
		ELSIF _GroupController.Enabled THEN
			_MoverCommander.ActivateTrack(_XtsSystem.Movers, XtsCoreParameters.InitialTrackId);
			_State := 51;
		END_IF

	51:
		//Add all to Track
		IF _MoverCommander.Error THEN
			_Error				 := TRUE;
			LogSource.SourceName := 'EnableXtsTask';
			LogMessage.Message	 := 'Failed to Activate to Track.';
			LogMessage.MessageId := E_XtsLogMessage.SystemEnableActivateTrackFailed;
			LogMessage.Severity	 := 3;
			_Logger.LogMessageInstance(LogSource, LogMessage);
			_ErrorId := _MoverCommander.ErrorId;
			_State	 := 255;
		ELSIF NOT _MoverCommander.Busy THEN
			_State := 60;
		END_IF

	60:
		//Enable All Stations
		IF NOT _XtsSystem.Config.CommandStationsOnEnable THEN
			LogSource.SourceName := 'EnableXtsTask';
			LogMessage.Message	 := 'Station Enable Skipped due to configuration.';
			LogMessage.MessageId := E_XtsLogMessage.SystemEnableActivateTrackFailed;
			LogMessage.Severity	 := 0;
			_Logger.LogMessageInstance(LogSource, LogMessage);
			_State := 70;
			RETURN;
		END_IF

		_StationCollection.ResetIterator();
		_Check := TRUE;
		WHILE _StationCollection.MoveToNext DO
			_StationCollection.Current.Enable();
			_Check := _Check AND _StationCollection.Current.Enabled;
		END_WHILE

		IF _Check THEN
			_State := 70;
		END_IF

	70:
		IF NOT _XtsSystem.Config.CommandPositionTriggersOnEnable THEN
			LogSource.SourceName := 'EnableXtsTask';
			LogMessage.Message	 := 'PositionTrigger Enable Skipped due to configuration.';
			LogMessage.MessageId := E_XtsLogMessage.SystemEnablePositionTriggerSkipped;
			LogMessage.Severity	 := 0;
			_Logger.LogMessageInstance(LogSource, LogMessage);
			_State := 80;
			RETURN;
		END_IF
		//Enable All Position Triggers
		_PositionTriggerCollection.ResetIterator();
		_Check := TRUE;
		WHILE _PositionTriggerCollection.MoveToNext DO
			_PositionTriggerCollection.Current.Enable();
			_Check := _Check AND _PositionTriggerCollection.Current.Enabled;
		END_WHILE

		IF _Check THEN
			_State := 80;
		END_IF
	80:
		LogSource.SourceName := 'EnableXtsTask';
		LogMessage.Message	 := 'XtsSystem Enabled.';
		LogMessage.MessageId := E_XtsLogMessage.SystemInfo;
		LogMessage.Severity	 := 1;
		_Logger.LogMessageInstance(LogSource, LogMessage);
		_Busy  := FALSE;
		_State := 81;
	81:
		IF NOT _CommandExecuted THEN
			_State := 0;
		END_IF
END_CASE
END_METHOD

METHOD Execute : I_XtsTaskResult
Execute			:= THIS^;
ExecuteWatchdog := ExecuteWatchdog + 1;
IF _CommandExecuted THEN
	RETURN;
END_IF

_CommandExecuted := TRUE;
_Busy			 := TRUE;
END_METHOD

//FB_Init is always available implicitly and it is used primarily for initialization.

//The return value is not evaluated. For a specific influence, you can also declare the

//methods explicitly and provide additional code there with the standard initialization

//code. You can evaluate the return value.
METHOD FB_Init : BOOL
VAR_INPUT
	bInitRetains		  : BOOL; // TRUE: the retain variables are initialized (reset warm / reset cold)
	bInCopyCode			  : BOOL; // TRUE: the instance will be copied to the copy code afterward (online change)
END_VAR
_TaskName := 'Enable Xts';
_TaskId	  := XtsSystemTaskId.ENABLE;
END_METHOD

METHOD Reset
_State			 := 0;
_Error			 := FALSE;
_ErrorId		 := 0;
_Busy			 := FALSE;
_CommandExecuted := FALSE;
END_METHOD

{attribute 'monitoring' := 'call'}
PROPERTY XpuId : I_XtsXpuId
GET
XpuId := _XpuId;
END_GET
SET
_XpuId := XpuId;
__QUERYINTERFACE(_XpuId, _XtsSystem);
__QUERYINTERFACE(_XtsSystem.Parameters, _CollisionAvoidanceGroupParameters);
__QUERYINTERFACE(_XpuId, _XtsStatus);
__QUERYINTERFACE(_XtsSystem.TracePublisher,_Logger);
_StationCollection		   := _XtsSystem.Stations;
_PositionTriggerCollection := _XtsSystem.PositionTriggers;
_ZoneCollection			   := _XtsSystem.Zones;
__QUERYINTERFACE(_XtsSystem.XtsTasks.GetTaskById(XtsSystemTaskId.MOVER_IDENTIFICATION), _MoverIdTask);
END_SET
END_PROPERTY

PROPERTY XtsMoverCommander : I_XtsMoverCommander
SET
_MoverCommander := XtsMoverCommander;
END_SET
END_PROPERTY

PROPERTY XtsMoverGroupController : I_XtsMoverGroupController
SET
_GroupController := XtsMoverGroupController;
END_SET
END_PROPERTY

END_FUNCTION_BLOCK

// _Internal/XtsSystem/Base/XtsTaskResult
{attribute 'no_explicit_call' := 'This FB is a CLASS and must be accessed using methods or properties'}
FUNCTION_BLOCK XtsTaskResult EXTENDS BaseTaskResult IMPLEMENTS I_XtsTaskResult
VAR
	_CommandExecuted : BOOL;
	_TaskId			 : XtsSystemTaskId;
	_Logger			 : I_XtsLogger;
END_VAR

{attribute 'monitoring':='call'}
PROPERTY TaskId : XtsSystemTaskId
GET
TaskId := _TaskId;
END_GET
END_PROPERTY

END_FUNCTION_BLOCK

// _Internal/XtsSystem/Tasks/Interfaces/I_XtsEnableTask
INTERFACE I_XtsEnableTask EXTENDS I_XtsTask, I_XtsExecutableTask, I_ContainXtsMoverCommander, I_ContainXtsMoverGroupController, I_Resettable

PROPERTY AxesGroup : REFERENCE TO AXES_GROUP_REF
GET
END_GET
SET
END_SET
END_PROPERTY

END_INTERFACE

// _Internal/XtsSystem/Tasks/Interfaces/I_XtsExecutableTask
INTERFACE I_XtsExecutableTask EXTENDS I_XtsTask

METHOD Execute : I_XtsTaskResult
END_METHOD

END_INTERFACE

// XtsMoverCommander/Interfaces/I_ContainXtsMoverCommander
INTERFACE I_ContainXtsMoverCommander EXTENDS I_Base

PROPERTY XtsMoverCommander : I_XtsMoverCommander
SET
END_SET
END_PROPERTY

END_INTERFACE

// XtsMoverCommander/XtsMoverCommander
{attribute 'hide_all_locals'}
FUNCTION_BLOCK XtsMoverCommander IMPLEMENTS I_XtsMoverCommander
VAR
	_CurrentCommand	 : I_XtsMoverTaskResult := NullObjects.XtsMoverTaskResult;
	_Enable			 : XtsMoverEnabler;
	_Disable		 : XtsMoverDisabler;
	_MoveToPosition	 : XtsMoverMoveToPosition;
	_MoveVelocity	 : XtsMoverMoveVelocity;
	_MoveToStation	 : XtsMoverMoveToStation;
	_ActivateTrack	 : XtsMoverActivateTrack;
	_Halt			 : XtsMoverHalt;
	_AddToGroup		 : XtsMoverAddToGroup;
	_RemoveFromGroup : XtsMoverRemoveFromGroup;
	_ParameterSet	 : XtsParameterSet;
END_VAR

//Command Mover to Activate to track
METHOD ActivateTrack : I_XtsMoverTaskResult
VAR_INPUT
	Visitee : I_AcceptXtsMoverVisitors;
	//Track to Activate to
	TrackId : UDINT; 
END_VAR
_ActivateTrack.TrackId		   := TrackId;
_ActivateTrack.ExecuteOn(Visitee);
_CurrentCommand := _ActivateTrack;
ActivateTrack	:= _CurrentCommand;
END_METHOD

//Add Mover to CA Group
METHOD AddToGroup: I_XtsMoverTaskResult
VAR_INPUT
	Visitee : I_AcceptXtsMoverVisitors;
	Group : REFERENCE TO AXES_GROUP_REF; //Group to Add to
	Ident : UDINT; //Ident in Group
END_VAR
_AddToGroup.AxesGroup		REF= Group;
_AddToGroup.IdentInGroup	:= Ident;
_AddToGroup.ExecuteOn(Visitee);
_CurrentCommand := _AddToGroup;
AddToGroup		:= _CurrentCommand;
END_METHOD

METHOD Disable : I_XtsMoverTaskResult
VAR_INPUT
	Visitee : I_AcceptXtsMoverVisitors;
END_VAR
_Disable.ExecuteOn(Visitee);
_CurrentCommand := _Disable;
Disable			:= _CurrentCommand;
END_METHOD

METHOD Enable : I_XtsMoverTaskResult
VAR_INPUT
	Visitee : I_AcceptXtsMoverVisitors;
END_VAR
_Enable.ExecuteOn(Visitee);
_CurrentCommand := _Enable;
Enable			:= _CurrentCommand;
END_METHOD

//Command Mover(s) to Halt
METHOD Halt : I_XtsMoverTaskResult
VAR_INPUT
	Visitee : I_AcceptXtsMoverVisitors;

	//Rate to Decelerate
	Deceleration : LREAL;

	//Gap to maintain to other movers
	Gap : LREAL;
END_VAR
_ParameterSet.Deceleration := Deceleration;
_ParameterSet.Gap		   := Gap;
_Halt.Deceleration		   := _ParameterSet.Deceleration;
_Halt.Gap				   := _ParameterSet.Gap;
_Halt.Jerk                 := _ParameterSet.Jerk;
_Halt.ExecuteOn(Visitee);
_CurrentCommand := _Halt;
Halt := _CurrentCommand;
END_METHOD

(*Command all Movers in Collection to Move To Position*)
METHOD MoveToPosition : I_XtsMoverTaskResult
VAR_INPUT
	Visitee : I_AcceptXtsMoverVisitors;
	(*Position to move to*)
	Position	: LREAL;
	(*Direction to move*)
	Direction	: Tc3_Mc3Definitions.MC_DIRECTION := Tc3_Mc3Definitions.MC_DIRECTION.mcDirectionPositive;
END_VAR
_MoveToPosition.Position		:= Position;
_MoveToPosition.Direction		:= Direction;
_MoveToPosition.Velocity		:= _ParameterSet.Velocity;
_MoveToPosition.Acceleration	:= _ParameterSet.Acceleration;
_MoveToPosition.Deceleration	:= _ParameterSet.Deceleration;
_MoveToPosition.Jerk			:= _ParameterSet.Jerk;
_MoveToPosition.Gap				:= _ParameterSet.Gap;
_MoveToPosition.Direction		:= _ParameterSet.Direction;
_MoveToPosition.ExecuteOn(Visitee);
_CurrentCommand := _MoveToPosition;
MoveToPosition	:= _CurrentCommand;
END_METHOD

(*Command all Movers in Collection to MoveToStation*)
METHOD MoveToStation : I_XtsMoverTaskResult
VAR_INPUT
	Visitee : I_AcceptXtsMoverVisitors;
	(*Station to move to*)
	Station	: I_XtsStation;
END_VAR
_MoveToStation.Station		:= Station;
_MoveToStation.Velocity		:= _ParameterSet.Velocity;
_MoveToStation.Acceleration := _ParameterSet.Acceleration;
_MoveToStation.Deceleration := _ParameterSet.Deceleration;
_MoveToStation.Jerk			:= _ParameterSet.Jerk;
_MoveToStation.Gap			:= _ParameterSet.Gap;
_MoveToStation.Direction	:= _ParameterSet.Direction;
_MoveToStation.ExecuteOn(Visitee);
_CurrentCommand := _MoveToStation;
MoveToStation	:= _CurrentCommand;
END_METHOD

(*Command all Movers in Collection to Move To Position*)
METHOD MoveVelocity : I_XtsMoverTaskResult
VAR_INPUT
	Visitee : I_AcceptXtsMoverVisitors;
	(*Velocity to move at*)
	Velocity	: LREAL;
	(*Direction to move*)
	Direction	: Tc3_Mc3Definitions.MC_DIRECTION := Tc3_Mc3Definitions.MC_DIRECTION.mcDirectionPositive;
END_VAR
_ParameterSet.Direction		  := Direction;
_ParameterSet.Velocity		  := Velocity;
_MoveVelocity.Velocity		  := _ParameterSet.Velocity;
_MoveVelocity.Acceleration	  := _ParameterSet.Acceleration;
_MoveVelocity.Deceleration	  := _ParameterSet.Deceleration;
_MoveVelocity.Jerk			  := _ParameterSet.Jerk;
_MoveVelocity.Gap			  := _ParameterSet.Gap;
_MoveVelocity.Direction		  := _ParameterSet.Direction;
_MoveVelocity.ExecuteOn(Visitee);
_CurrentCommand := _MoveVelocity;
MoveVelocity	:= _CurrentCommand;
END_METHOD

//Remove Mover From CA Group
METHOD RemoveFromGroup: I_XtsMoverTaskResult
VAR_INPUT
	Visitee : I_AcceptXtsMoverVisitors;
	Group : REFERENCE TO AXES_GROUP_REF; //Group to Remove from
	Ident : UDINT; //Ident in Group
END_VAR
_RemoveFromGroup.AxesGroup		 REF= Group;
_RemoveFromGroup.IdentInGroup	 := Ident;
_RemoveFromGroup.ExecuteOn(Visitee);
_CurrentCommand := _RemoveFromGroup;
RemoveFromGroup := _CurrentCommand;
END_METHOD

{attribute 'monitoring':='call'}
PROPERTY Busy : BOOL
GET
Busy := _CurrentCommand.Busy;
END_GET
END_PROPERTY

{attribute 'monitoring':='call'}
PROPERTY CurrentTask : I_XtsMoverTaskResult
GET
CurrentTask := _CurrentCommand;
END_GET
END_PROPERTY

{attribute 'monitoring':='call'}
PROPERTY Error : BOOL
GET
Error := _CurrentCommand.Error;
END_GET
END_PROPERTY

{attribute 'monitoring':='call'}
PROPERTY ErrorId : UDINT
GET
ErrorId := _CurrentCommand.ErrorId;
END_GET
END_PROPERTY

{attribute 'monitoring' := 'call'}
PROPERTY Parameters : I_XtsParameterSet
GET
Parameters := _ParameterSet;
END_GET
SET
_ParameterSet.CopyFrom(Parameters);
END_SET
END_PROPERTY

{attribute 'monitoring' := 'call'}
PROPERTY TaskName : STRING
GET
TaskName := _CurrentCommand.TaskName;
END_GET
END_PROPERTY

END_FUNCTION_BLOCK

// XtsMoverCommander/Interfaces/I_XtsMoverCommander
INTERFACE I_XtsMoverCommander EXTENDS I_Base, I_HasXtsParameters, I_TaskResult

//Command Mover to Activate to track
METHOD ActivateTrack : I_XtsMoverTaskResult
VAR_INPUT
	Visitee : I_AcceptXtsMoverVisitors;
	//Track to Activate to
	TrackId : UDINT; 
END_VAR
END_METHOD

//Add Mover to CA Group
METHOD AddToGroup: I_XtsMoverTaskResult
VAR_INPUT
	Visitee : I_AcceptXtsMoverVisitors;
	Group : REFERENCE TO AXES_GROUP_REF; //Group to Add to
	Ident : UDINT; //Ident in Group
END_VAR
END_METHOD

METHOD Disable : I_XtsMoverTaskResult
VAR_INPUT
	Visitee : I_AcceptXtsMoverVisitors;
END_VAR
END_METHOD

METHOD Enable : I_XtsMoverTaskResult
VAR_INPUT
	Visitee : I_AcceptXtsMoverVisitors;
END_VAR
END_METHOD

//Command Mover(s) to Halt
METHOD Halt : I_XtsMoverTaskResult
VAR_INPUT
	Visitee : I_AcceptXtsMoverVisitors;

	//Rate to Decelerate
	Deceleration : LREAL;

	//Gap to maintain to other movers
	Gap : LREAL;
END_VAR
END_METHOD

(*Command all Movers in Collection to Move To Position*)
METHOD MoveToPosition : I_XtsMoverTaskResult
VAR_INPUT
	Visitee : I_AcceptXtsMoverVisitors;
	(*Position to move to*)
	Position	: LREAL;
	(*Direction to move*)
	Direction	: Tc3_Mc3Definitions.MC_DIRECTION := Tc3_Mc3Definitions.MC_DIRECTION.mcDirectionPositive;
END_VAR
END_METHOD

(*Command all Movers in Collection to MoveToStation*)
METHOD MoveToStation : I_XtsMoverTaskResult
VAR_INPUT
	Visitee : I_AcceptXtsMoverVisitors;

	(*Station to move to*)
	Station : I_XtsStation;
END_VAR
END_METHOD

(*Command all Movers in Collection to Move To Position*)
METHOD MoveVelocity : I_XtsMoverTaskResult
VAR_INPUT
	Visitee : I_AcceptXtsMoverVisitors;
	(*Velocity to move at*)
	Velocity	: LREAL;
	(*Direction to move*)
	Direction	: Tc3_Mc3Definitions.MC_DIRECTION := Tc3_Mc3Definitions.MC_DIRECTION.mcDirectionPositive;
END_VAR
END_METHOD

//Remove Mover From CA Group
METHOD RemoveFromGroup: I_XtsMoverTaskResult
VAR_INPUT
	Visitee : I_AcceptXtsMoverVisitors;
	Group : REFERENCE TO AXES_GROUP_REF; //Group to Remove from
	Ident : UDINT; //Ident in Group
END_VAR
END_METHOD

END_INTERFACE

// _Internal/Mover/MoverTaskBase/XtsMoverTaskResult
{attribute 'no_explicit_call' := 'This FB is a CLASS and must be accessed using methods or properties'}
FUNCTION_BLOCK XtsMoverTaskResult EXTENDS BaseTaskResult IMPLEMENTS I_Cyclic
VAR
	_TaskId			 : MoverTaskID;
	_Aborted		 : BOOL;
	_Mover			 : I_XtsMover;
	_CommandExecuted : BOOL;
	WatchdogCheck	 : UDINT;
	ExecuteWatchdog	 : UDINT;
	{attribute 'hide'}
	_Logger : I_XtsLogger;
	{attribute 'hide'}
	LogSource : TraceSourceInfo;
	{attribute 'hide'}
	LogMessage : TraceMessageInfo;
END_VAR

{attribute 'monitoring' := 'call'}
PROPERTY Aborted : BOOL
GET
Aborted := _Aborted;
END_GET
END_PROPERTY

PROPERTY CommandExecuted : BOOL
GET
CommandExecuted := _CommandExecuted;
END_GET
END_PROPERTY

METHOD CyclicLogic
IF ExecuteWatchdog <> WatchdogCheck THEN
	WatchdogCheck := ExecuteWatchdog;
ELSE
	ExecuteWatchdog	 := 0;
	_CommandExecuted := FALSE;
END_IF
END_METHOD

PROPERTY Mover : I_XtsMover
SET
_Mover := Mover;
END_SET
END_PROPERTY

{attribute 'monitoring':='call'}
PROPERTY TaskId : MoverTaskId
GET
TaskId := _TaskId;
END_GET
END_PROPERTY

END_FUNCTION_BLOCK

// MoverVisitors/XtsMoverEnabler
FUNCTION_BLOCK XtsMoverEnabler IMPLEMENTS I_XtsMoverVisitor, I_XtsMoverTaskResult, I_XtsMoverVisitorTask
VAR
	_Status		  : Collection<XtsCoreParameters.MaxNumberOfMovers>;
	_Visitee	  : I_AcceptXtsMoverVisitors;
END_VAR

{attribute 'monitoring':='call'}
PROPERTY XtsMoverVisitee : I_AcceptXtsMoverVisitors
GET
XtsMoverVisitee := _Visitee;
END_GET
SET
_Visitee := XtsMoverVisitee;
END_SET
END_PROPERTY

{attribute 'monitoring' := 'call'}
PROPERTY Aborted : BOOL
GET
Aborted := FALSE;
END_GET
END_PROPERTY

{attribute 'monitoring':='call'}
PROPERTY Busy : BOOL
GET
VAR
	Status : I_XtsMover;
END_VAR
_Status.ResetIterator();
WHILE _Status.MoveToNext DO
	__QUERYINTERFACE(_Status.Current, Status);
	IF Status.CurrentTask.Busy THEN
		Busy := TRUE;
		RETURN;
	END_IF
END_WHILE
END_GET
END_PROPERTY

PROPERTY CommandExecuted : BOOL
GET
VAR
	Status : I_XtsMoverTaskResult;
END_VAR
_Status.ResetIterator();
WHILE _Status.MoveToNext DO
	__QUERYINTERFACE(_Status.Current, Status);
	IF Status.CommandExecuted THEN
		CommandExecuted := TRUE;
		RETURN;
	END_IF
END_WHILE
END_GET
END_PROPERTY

{attribute 'monitoring':='call'}
PROPERTY Error : BOOL
GET
VAR
	Status : I_XtsMover;
END_VAR
_Status.ResetIterator();
WHILE _Status.MoveToNext DO
	__QUERYINTERFACE(_Status.Current, Status);
	IF Status.CurrentTask.Error THEN
		Error := TRUE;
		RETURN;
	END_IF
END_WHILE
END_GET
END_PROPERTY

{attribute 'monitoring':='call'}
PROPERTY ErrorId : UDINT
GET
VAR
	Status : I_XtsMover;
END_VAR
_Status.ResetIterator();
WHILE _Status.MoveToNext DO
	__QUERYINTERFACE(_Status.Current, Status);
	IF Status.CurrentTask.Error THEN
		ErrorId := Status.CurrentTask.ErrorId;
		RETURN;
	END_IF
END_WHILE
END_GET
END_PROPERTY

METHOD ExecuteOn : I_XtsMoverTaskResult
VAR_INPUT
	Visitee  : I_AcceptXtsMoverVisitors;
END_VAR
_Status.Clear();
_Visitee := Visitee;
_Visitee.AcceptMoverVisitor(THIS^);
ExecuteOn := THIS^;
END_METHOD

{attribute 'monitoring' := 'call'}
PROPERTY TaskId : MoverTaskId
GET
TaskId := MoverTaskId.ENABLE;
END_GET
END_PROPERTY

{attribute 'monitoring' := 'call'}
PROPERTY TaskName : STRING
GET
TaskName := 'Enable Mover';
END_GET
END_PROPERTY

METHOD VisitMover
VAR_INPUT
	Mover	: I_XtsMover;
END_VAR
Mover.Enable();
_Status.AddItem(Mover);
END_METHOD

END_FUNCTION_BLOCK

// MoverVisitors/Interfaces/I_XtsMoverVisitorTask
INTERFACE I_XtsMoverVisitorTask EXTENDS I_Base

METHOD ExecuteOn : I_XtsMoverTaskResult
VAR_INPUT
	Visitee : I_AcceptXtsMoverVisitors;
END_VAR
END_METHOD

END_INTERFACE

// MoverVisitors/XtsMoverDisabler
FUNCTION_BLOCK XtsMoverDisabler IMPLEMENTS I_XtsMoverVisitor, I_XtsMoverTaskResult, I_XtsMoverVisitorTask
VAR
	_Status		  : Collection<XtsCoreParameters.MaxNumberOfMovers>;
	_Visitee	  : I_AcceptXtsMoverVisitors;
END_VAR

{attribute 'monitoring':='call'}
PROPERTY XtsMoverVisitee : I_AcceptXtsMoverVisitors
GET
XtsMoverVisitee := _Visitee;
END_GET
SET
_Visitee := XtsMoverVisitee;
END_SET
END_PROPERTY

{attribute 'monitoring' := 'call'}
PROPERTY Aborted : BOOL
GET
Aborted := FALSE;
END_GET
END_PROPERTY

{attribute 'monitoring':='call'}
PROPERTY Busy : BOOL
GET
VAR
	Status : I_XtsMover;
END_VAR
_Status.ResetIterator();
WHILE _Status.MoveToNext DO
	__QUERYINTERFACE(_Status.Current, Status);
	IF Status.CurrentTask.Busy THEN
		Busy := TRUE;
		RETURN;
	END_IF
END_WHILE
END_GET
END_PROPERTY

PROPERTY CommandExecuted : BOOL
GET
VAR
	Status : I_XtsMoverTaskResult;
END_VAR
_Status.ResetIterator();
WHILE _Status.MoveToNext DO
	__QUERYINTERFACE(_Status.Current, Status);
	IF Status.CommandExecuted THEN
		CommandExecuted := TRUE;
		RETURN;
	END_IF
END_WHILE
END_GET
END_PROPERTY

{attribute 'monitoring':='call'}
PROPERTY Error : BOOL
GET
VAR
	Status : I_XtsMover;
END_VAR
_Status.ResetIterator();
WHILE _Status.MoveToNext DO
	__QUERYINTERFACE(_Status.Current, Status);
	IF Status.CurrentTask.Error THEN
		Error := TRUE;
		RETURN;
	END_IF
END_WHILE
END_GET
END_PROPERTY

{attribute 'monitoring':='call'}
PROPERTY ErrorId : UDINT
GET
VAR
	Status : I_XtsMover;
END_VAR
_Status.ResetIterator();
WHILE _Status.MoveToNext DO
	__QUERYINTERFACE(_Status.Current, Status);
	IF Status.CurrentTask.Error THEN
		ErrorId := Status.CurrentTask.ErrorId;
		RETURN;
	END_IF
END_WHILE
END_GET
END_PROPERTY

METHOD ExecuteOn : I_XtsMoverTaskResult
VAR_INPUT
	Visitee  : I_AcceptXtsMoverVisitors;
END_VAR
_Status.Clear();
_Visitee := Visitee;
_Visitee.AcceptMoverVisitor(THIS^);
ExecuteOn := THIS^;
END_METHOD

{attribute 'monitoring' := 'call'}
PROPERTY TaskId : MoverTaskId
GET
TaskId := MoverTaskId.DISABLE;
END_GET
END_PROPERTY

{attribute 'monitoring' := 'call'}
PROPERTY TaskName : STRING
GET
TaskName := 'Disable Mover';
END_GET
END_PROPERTY

METHOD VisitMover
VAR_INPUT
	Mover	: I_XtsMover;
END_VAR
Mover.Disable();
_Status.AddItem(Mover);
END_METHOD

END_FUNCTION_BLOCK

// MoverVisitors/XtsMoverMoveToPosition
FUNCTION_BLOCK XtsMoverMoveToPosition IMPLEMENTS I_XtsMoverVisitor, I_BaseDynamics, I_CollisionAvoidanceDynamics, I_MoveToPositionParameters, I_XtsMoverTaskResult, I_XtsMoverVisitorTask
VAR
	_Status		   : Collection<XtsCoreParameters.MaxNumberOfMovers>;
	_Visitee	   : I_AcceptXtsMoverVisitors;
	_Dynamics	   : BaseDynamics;
	_Position	   : MoveToPositionParameters;
	_Gap		   : CollisionAvoidanceDynamics;
END_VAR

{attribute 'monitoring' := 'call'}
PROPERTY Acceleration : LREAL
GET
Acceleration := _Dynamics.Acceleration;
END_GET
SET
_Dynamics.Acceleration := Acceleration;
END_SET
END_PROPERTY

METHOD CopyParametersFrom
VAR_INPUT
	CopyFrom : I_XtsParameterSet;
END_VAR
_Dynamics.Velocity	   := CopyFrom.Velocity;
_Dynamics.Acceleration := CopyFrom.Acceleration;
_Dynamics.Deceleration := CopyFrom.Deceleration;
_Dynamics.Jerk		   := CopyFrom.Jerk;
_Dynamics.Direction	   := CopyFrom.Direction;
_Position.Position	   := CopyFrom.Position;
_Gap.Gap			   := CopyFrom.Gap;
END_METHOD

{attribute 'monitoring' := 'call'}
PROPERTY Deceleration : LREAL
GET
Deceleration := _Dynamics.Deceleration;
END_GET
SET
_Dynamics.Deceleration := Deceleration;
END_SET
END_PROPERTY

{attribute 'monitoring' := 'call'}
PROPERTY Direction : Tc3_Mc3Definitions.MC_DIRECTION
GET
Direction := _Dynamics.Direction;
END_GET
SET
_Dynamics.Direction := Direction;
END_SET
END_PROPERTY

{attribute 'monitoring' := 'call'}
PROPERTY Gap : LREAL
GET
Gap := _Gap.Gap;
END_GET
SET
_Gap.Gap := Gap;
END_SET
END_PROPERTY

{attribute 'monitoring' := 'call'}
PROPERTY Jerk : LREAL
GET
Jerk := _Dynamics.Jerk;
END_GET
SET
_Dynamics.Jerk := Jerk;
END_SET
END_PROPERTY

{attribute 'monitoring' := 'call'}
PROPERTY Position : LREAL
GET
Position := _Position.Position;
END_GET
SET
_Position.Position := Position;
END_SET
END_PROPERTY

{attribute 'monitoring' := 'call'}
PROPERTY Velocity : LREAL
GET
Velocity := _Dynamics.Velocity;
END_GET
SET
_Dynamics.Velocity := Velocity;
END_SET
END_PROPERTY

{attribute 'monitoring':='call'}
PROPERTY XtsMoverVisitee : I_AcceptXtsMoverVisitors
GET
XtsMoverVisitee := _Visitee;
END_GET
SET
_Visitee := XtsMoverVisitee;
END_SET
END_PROPERTY

{attribute 'monitoring' := 'call'}
PROPERTY Aborted : BOOL
GET
END_GET
END_PROPERTY

{attribute 'monitoring':='call'}
PROPERTY Busy : BOOL
GET
VAR
	Status : I_XtsMoverTaskResult;
END_VAR
_Status.ResetIterator();
WHILE _Status.MoveToNext DO
	__QUERYINTERFACE(_Status.Current, Status);
	IF Status.Busy THEN
		Busy := TRUE;
		RETURN;
	END_IF
END_WHILE
END_GET
END_PROPERTY

PROPERTY CommandExecuted : BOOL
GET
VAR
	Status : I_XtsMoverTaskResult;
END_VAR
_Status.ResetIterator();
WHILE _Status.MoveToNext DO
	__QUERYINTERFACE(_Status.Current, Status);
	IF Status.CommandExecuted THEN
		CommandExecuted := TRUE;
		RETURN;
	END_IF
END_WHILE
END_GET
END_PROPERTY

{attribute 'monitoring':='call'}
PROPERTY Error : BOOL
GET
VAR
	Status : I_XtsMoverTaskResult;
END_VAR
_Status.ResetIterator();
WHILE _Status.MoveToNext DO
	__QUERYINTERFACE(_Status.Current, Status);
	IF Status.Error THEN
		Error := TRUE;
		RETURN;
	END_IF
END_WHILE
END_GET
END_PROPERTY

{attribute 'monitoring':='call'}
PROPERTY ErrorId : UDINT
GET
VAR
	Status : I_XtsMoverTaskResult;
END_VAR
_Status.ResetIterator();
WHILE _Status.MoveToNext DO
	__QUERYINTERFACE(_Status.Current, Status);
	IF Status.Error THEN
		ErrorId := Status.ErrorId;
		RETURN;
	END_IF
END_WHILE
END_GET
END_PROPERTY

METHOD ExecuteOn : I_XtsMoverTaskResult
VAR_INPUT
	Visitee : I_AcceptXtsMoverVisitors;
END_VAR
_Status.Clear();
_Visitee := Visitee;
_Visitee.AcceptMoverVisitor(THIS^);
ExecuteOn := THIS^;
END_METHOD

{attribute 'monitoring' := 'call'}
PROPERTY TaskId : MoverTaskId
GET
TaskId := MoverTaskId.MOVE_TO_POSITION;
END_GET
END_PROPERTY

{attribute 'monitoring' := 'call'}
PROPERTY TaskName : STRING
GET
TaskName := 'Move To Position';
END_GET
END_PROPERTY

METHOD VisitMover
VAR_INPUT
	Mover	: I_XtsMover;
END_VAR
VAR
	Result : I_XtsMoverTaskResult;
END_VAR
Mover.Parameters.Velocity	  := _Dynamics.Velocity;
Mover.Parameters.Acceleration := _Dynamics.Acceleration;
Mover.Parameters.Deceleration := _Dynamics.Deceleration;
Mover.Parameters.Jerk		  := _Dynamics.Jerk;
Mover.Parameters.Gap		  := _Gap.Gap;
Result						  := Mover.MoveToPosition(Position := _Position.Position, Direction := _Dynamics.Direction);
_Status.AddItem(Result);
END_METHOD

END_FUNCTION_BLOCK

// _Internal/Mover/Parameters/BaseDynamics
{attribute 'no_explicit_call' := 'This FB is a CLASS and must be accessed using methods or properties'}
FUNCTION_BLOCK BaseDynamics IMPLEMENTS I_BaseDynamics
VAR
	_Acceleration : LREAL;
	_Deceleration : LREAL;
	_Direction	  : Tc3_Mc3Definitions.MC_DIRECTION := Tc3_Mc3Definitions.MC_DIRECTION.mcDirectionPositive;
	_Velocity	  : LREAL;
	_Jerk		  : LREAL;
END_VAR

{attribute 'monitoring' := 'call'}
PROPERTY Acceleration : LREAL
GET
Acceleration := _Acceleration;
END_GET
SET
_Acceleration := Acceleration;
END_SET
END_PROPERTY

{attribute 'monitoring' := 'call'}
PROPERTY Deceleration : LREAL
GET
Deceleration := _Deceleration;
END_GET
SET
_Deceleration := Deceleration;
END_SET
END_PROPERTY

{attribute 'monitoring' := 'call'}
PROPERTY Direction : Tc3_Mc3Definitions.MC_DIRECTION
GET
Direction := _Direction;
END_GET
SET
_Direction := Direction;
END_SET
END_PROPERTY

{attribute 'monitoring' := 'call'}
PROPERTY Jerk : LREAL
GET
Jerk := _Jerk;
END_GET
SET
_Jerk := Jerk;
END_SET
END_PROPERTY

{attribute 'monitoring' := 'call'}
PROPERTY Velocity : LREAL
GET
Velocity := _Velocity;
END_GET
SET
_Velocity := Velocity;
END_SET
END_PROPERTY

END_FUNCTION_BLOCK

// _Internal/Mover/Parameters/MoveToPositionParameters
{attribute 'no_explicit_call' := 'This FB is a CLASS and must be accessed using methods or properties'}
FUNCTION_BLOCK MoveToPositionParameters IMPLEMENTS I_MoveToPositionParameters
VAR
	_CommandedPosition : LREAL := 0;
END_VAR

{attribute 'monitoring' := 'call'}
PROPERTY Position : LREAL
GET
Position := _CommandedPosition;
END_GET
SET
_CommandedPosition := Position;
END_SET
END_PROPERTY

END_FUNCTION_BLOCK

// _Internal/Mover/Parameters/CollisionAvoidanceDynamics
{attribute 'no_explicit_call' := 'This FB is a CLASS and must be accessed using methods or properties'}
FUNCTION_BLOCK CollisionAvoidanceDynamics IMPLEMENTS I_CollisionAvoidanceDynamics
VAR
	_Gap : LREAL;
END_VAR

{attribute 'monitoring' := 'call'}
PROPERTY Gap : LREAL
GET
Gap := _Gap;
END_GET
SET
_Gap := Gap;
END_SET
END_PROPERTY

END_FUNCTION_BLOCK

// MoverVisitors/XtsMoverMoveVelocity
FUNCTION_BLOCK XtsMoverMoveVelocity IMPLEMENTS I_XtsMoverVisitor, I_BaseDynamics, I_CollisionAvoidanceDynamics, I_XtsMoverTaskResult, I_XtsMoverVisitorTask
VAR
	_Status		   : Collection<XtsCoreParameters.MaxNumberOfMovers>;
	_Visitee	   : I_AcceptXtsMoverVisitors;
	_Dynamics	   : BaseDynamics;
	_Gap		   : CollisionAvoidanceDynamics;
END_VAR

{attribute 'monitoring' := 'call'}
PROPERTY Acceleration : LREAL
GET
Acceleration := _Dynamics.Acceleration;
END_GET
SET
_Dynamics.Acceleration := Acceleration;
END_SET
END_PROPERTY

METHOD CopyParametersFrom
VAR_INPUT
	CopyFrom : I_XtsParameterSet;
END_VAR
_Dynamics.Velocity	   := CopyFrom.Velocity;
_Dynamics.Acceleration := CopyFrom.Acceleration;
_Dynamics.Deceleration := CopyFrom.Deceleration;
_Dynamics.Direction	   := CopyFrom.Direction;
_Dynamics.Jerk		   := CopyFrom.Jerk;
_Gap.Gap			   := CopyFrom.Gap;
END_METHOD

{attribute 'monitoring' := 'call'}
PROPERTY Deceleration : LREAL
GET
Deceleration := _Dynamics.Deceleration;
END_GET
SET
_Dynamics.Deceleration := Deceleration;
END_SET
END_PROPERTY

{attribute 'monitoring' := 'call'}
PROPERTY Direction : Tc3_Mc3Definitions.MC_DIRECTION
GET
Direction := _Dynamics.Direction;
END_GET
SET
_Dynamics.Direction := Direction;
END_SET
END_PROPERTY

{attribute 'monitoring' := 'call'}
PROPERTY Gap : LREAL
GET
Gap := _Gap.Gap;
END_GET
SET
_Gap.Gap := Gap;
END_SET
END_PROPERTY

{attribute 'monitoring' := 'call'}
PROPERTY Jerk : LREAL
GET
Jerk := _Dynamics.Jerk;
END_GET
SET
_Dynamics.Jerk := Jerk;
END_SET
END_PROPERTY

{attribute 'monitoring' := 'call'}
PROPERTY Velocity : LREAL
GET
Velocity := _Dynamics.Velocity;
END_GET
SET
_Dynamics.Velocity := Velocity;
END_SET
END_PROPERTY

{attribute 'monitoring':='call'}
PROPERTY XtsMoverVisitee : I_AcceptXtsMoverVisitors
GET
XtsMoverVisitee := _Visitee;
END_GET
SET
_Visitee := XtsMoverVisitee;
END_SET
END_PROPERTY

{attribute 'monitoring' := 'call'}
PROPERTY Aborted : BOOL
GET
END_GET
END_PROPERTY

{attribute 'monitoring':='call'}
PROPERTY Busy : BOOL
GET
VAR
	Status : I_XtsMoverTaskResult;
END_VAR
_Status.ResetIterator();
WHILE _Status.MoveToNext DO
	__QUERYINTERFACE(_Status.Current, Status);
	IF Status.Busy THEN
		Busy := TRUE;
		RETURN;
	END_IF
END_WHILE
END_GET
END_PROPERTY

PROPERTY CommandExecuted : BOOL
GET
VAR
	Status : I_XtsMoverTaskResult;
END_VAR
_Status.ResetIterator();
WHILE _Status.MoveToNext DO
	__QUERYINTERFACE(_Status.Current, Status);
	IF Status.CommandExecuted THEN
		CommandExecuted := TRUE;
		RETURN;
	END_IF
END_WHILE
END_GET
END_PROPERTY

{attribute 'monitoring':='call'}
PROPERTY Error : BOOL
GET
VAR
	Status : I_XtsMoverTaskResult;
END_VAR
_Status.ResetIterator();
WHILE _Status.MoveToNext DO
	__QUERYINTERFACE(_Status.Current, Status);
	IF Status.Error THEN
		Error := TRUE;
		RETURN;
	END_IF
END_WHILE
END_GET
END_PROPERTY

{attribute 'monitoring':='call'}
PROPERTY ErrorId : UDINT
GET
VAR
	Status : I_XtsMoverTaskResult;
END_VAR
_Status.ResetIterator();
WHILE _Status.MoveToNext DO
	__QUERYINTERFACE(_Status.Current, Status);
	IF Status.Error THEN
		ErrorId := Status.ErrorId;
		RETURN;
	END_IF
END_WHILE
END_GET
END_PROPERTY

METHOD ExecuteOn : I_XtsMoverTaskResult
VAR_INPUT
	Visitee : I_AcceptXtsMoverVisitors;
END_VAR
_Status.Clear();
_Visitee := Visitee;
_Visitee.AcceptMoverVisitor(THIS^);
ExecuteOn := THIS^;
END_METHOD

{attribute 'monitoring' := 'call'}
PROPERTY TaskId : MoverTaskId
GET
TaskId := MoverTaskId.MOVE_VELOCITY;
END_GET
END_PROPERTY

{attribute 'monitoring' := 'call'}
PROPERTY TaskName : STRING
GET
TaskName := 'Move Velocity';
END_GET
END_PROPERTY

METHOD VisitMover
VAR_INPUT
	Mover	: I_XtsMover;
END_VAR
VAR
	Result : I_XtsMoverTaskResult;
END_VAR
Mover.Parameters.Acceleration := _Dynamics.Acceleration;
Mover.Parameters.Deceleration := _Dynamics.Deceleration;
Mover.Parameters.Jerk		  := _Dynamics.Jerk;
Mover.Parameters.Gap		  := _Gap.Gap;
Result						  := Mover.MoveVelocity(_Dynamics.Velocity, _Dynamics.Direction);
_Status.AddItem(Result);
END_METHOD

END_FUNCTION_BLOCK

// MoverVisitors/XtsMoverMoveToStation
FUNCTION_BLOCK XtsMoverMoveToStation IMPLEMENTS I_XtsMoverVisitor, I_BaseDynamics, I_CollisionAvoidanceDynamics, I_MoveToStationParameters, I_XtsMoverTaskResult, I_XtsMoverVisitorTask
VAR
	_Status		   : Collection<XtsCoreParameters.MaxNumberOfMovers>;
	_Visitee	   : I_AcceptXtsMoverVisitors;
	_Dynamics	   : BaseDynamics;
	_Station	   : MoveToStationParameters;
	_Gap		   : CollisionAvoidanceDynamics;
END_VAR

{attribute 'monitoring' := 'call'}
PROPERTY Acceleration : LREAL
GET
Acceleration := _Dynamics.Acceleration;
END_GET
SET
_Dynamics.Acceleration := Acceleration;
END_SET
END_PROPERTY

METHOD CopyParametersFrom
VAR_INPUT
	CopyFrom : I_XtsParameterSet;
END_VAR
_Dynamics.Velocity	   := CopyFrom.Velocity;
_Dynamics.Acceleration := CopyFrom.Acceleration;
_Dynamics.Deceleration := CopyFrom.Deceleration;
_Dynamics.Jerk		   := CopyFrom.Jerk;
_Dynamics.Direction	   := CopyFrom.Direction;
_Gap.Gap			   := CopyFrom.Gap;
END_METHOD

{attribute 'monitoring' := 'call'}
PROPERTY Deceleration : LREAL
GET
Deceleration := _Dynamics.Deceleration;
END_GET
SET
_Dynamics.Deceleration := Deceleration;
END_SET
END_PROPERTY

{attribute 'monitoring' := 'call'}
PROPERTY Direction : Tc3_Mc3Definitions.MC_DIRECTION
GET
Direction := _Dynamics.Direction;
END_GET
SET
_Dynamics.Direction := Direction;
END_SET
END_PROPERTY

{attribute 'monitoring' := 'call'}
PROPERTY Gap : LREAL
GET
Gap := _Gap.Gap;
END_GET
SET
_Gap.Gap := Gap;
END_SET
END_PROPERTY

{attribute 'monitoring' := 'call'}
PROPERTY Jerk : LREAL
GET
Jerk := _Dynamics.Jerk;
END_GET
SET
_Dynamics.Jerk := Jerk;
END_SET
END_PROPERTY

{attribute 'monitoring' := 'call'}
PROPERTY Station : I_XtsStation
GET
Station := _Station.Station;
END_GET
SET
_Station.Station := Station;
END_SET
END_PROPERTY

{attribute 'monitoring' := 'call'}
PROPERTY Velocity : LREAL
GET
Velocity := _Dynamics.Velocity;
END_GET
SET
_Dynamics.Velocity := Velocity;
END_SET
END_PROPERTY

{attribute 'monitoring':='call'}
PROPERTY XtsMoverVisitee : I_AcceptXtsMoverVisitors
GET
XtsMoverVisitee := _Visitee;
END_GET
SET
_Visitee := XtsMoverVisitee;
END_SET
END_PROPERTY

{attribute 'monitoring' := 'call'}
PROPERTY Aborted : BOOL
GET
END_GET
END_PROPERTY

{attribute 'monitoring':='call'}
PROPERTY Busy : BOOL
GET
VAR
	Status : I_XtsMoverTaskResult;
END_VAR
_Status.ResetIterator();
WHILE _Status.MoveToNext DO
	__QUERYINTERFACE(_Status.Current, Status);
	IF Status.Busy THEN
		Busy := TRUE;
		RETURN;
	END_IF
END_WHILE
END_GET
END_PROPERTY

PROPERTY CommandExecuted : BOOL
GET
VAR
	Status : I_XtsMoverTaskResult;
END_VAR
_Status.ResetIterator();
WHILE _Status.MoveToNext DO
	__QUERYINTERFACE(_Status.Current, Status);
	IF Status.CommandExecuted THEN
		CommandExecuted := TRUE;
		RETURN;
	END_IF
END_WHILE
END_GET
END_PROPERTY

{attribute 'monitoring':='call'}
PROPERTY Error : BOOL
GET
VAR
	Status : I_XtsMoverTaskResult;
END_VAR
_Status.ResetIterator();
WHILE _Status.MoveToNext DO
	__QUERYINTERFACE(_Status.Current, Status);
	IF Status.Error THEN
		Error := TRUE;
		RETURN;
	END_IF
END_WHILE
END_GET
END_PROPERTY

{attribute 'monitoring':='call'}
PROPERTY ErrorId : UDINT
GET
VAR
	Status : I_XtsMoverTaskResult;
END_VAR
_Status.ResetIterator();
WHILE _Status.MoveToNext DO
	__QUERYINTERFACE(_Status.Current, Status);
	IF Status.Error THEN
		ErrorId := Status.ErrorId;
		RETURN;
	END_IF
END_WHILE
END_GET
END_PROPERTY

METHOD ExecuteOn : I_XtsMoverTaskResult
VAR_INPUT
	Visitee : I_AcceptXtsMoverVisitors;
END_VAR
_Status.Clear();
_Visitee := Visitee;
_Visitee.AcceptMoverVisitor(THIS^);
ExecuteOn := THIS^;
END_METHOD

{attribute 'monitoring' := 'call'}
PROPERTY TaskId : MoverTaskId
GET
TaskId := MoverTaskId.MOVE_TO_STATION;
END_GET
END_PROPERTY

{attribute 'monitoring' := 'call'}
PROPERTY TaskName : STRING
GET
TaskName := 'Move To Station';
END_GET
END_PROPERTY

METHOD VisitMover
VAR_INPUT
	Mover	: I_XtsMover;
END_VAR
VAR
	Result : I_XtsMoverTaskResult;
END_VAR
Mover.Parameters.Velocity	  := _Dynamics.Velocity;
Mover.Parameters.Acceleration := _Dynamics.Acceleration;
Mover.Parameters.Deceleration := _Dynamics.Deceleration;
Mover.Parameters.Jerk		  := _Dynamics.Jerk;
Mover.Parameters.Direction	  := _Dynamics.Direction;
Mover.Parameters.Gap		  := _Gap.Gap;
Result						  := Mover.MoveToStation(Station := _Station.Station);
_Status.AddItem(Result);
END_METHOD

END_FUNCTION_BLOCK

// _Internal/Mover/Parameters/Interfaces/I_MoveToStationParameters
INTERFACE I_MoveToStationParameters EXTENDS I_Base

{attribute 'monitoring' := 'call'}
PROPERTY Station : I_XtsStation
GET
END_GET
SET
END_SET
END_PROPERTY

END_INTERFACE

// _Internal/Mover/Parameters/MoveToStationParameters
{attribute 'no_explicit_call' := 'This FB is a CLASS and must be accessed using methods or properties'}
FUNCTION_BLOCK MoveToStationParameters IMPLEMENTS I_MoveToStationParameters
VAR
	_DestinationStation : I_XtsStation := NullObjects.Station;
END_VAR

{attribute 'monitoring':='call'}
PROPERTY Station : I_XtsStation
GET
Station := _DestinationStation;
END_GET
SET
_DestinationStation := Station;
END_SET
END_PROPERTY

END_FUNCTION_BLOCK

// MoverVisitors/XtsMoverActivateTrack
FUNCTION_BLOCK XtsMoverActivateTrack IMPLEMENTS I_XtsMoverVisitor, I_XtsMoverTaskResult, I_XtsMoverVisitorTask
VAR
	_Status	 : Collection<XtsCoreParameters.MaxNumberOfMovers>;
	_Visitee : I_AcceptXtsMoverVisitors;
	_TrackId : UDINT;
END_VAR

METHOD CopyParametersFrom
VAR_INPUT
	CopyFrom : I_XtsParameterSet;
END_VAR
_TrackId := CopyFrom.Track.Id;
END_METHOD

{attribute 'monitoring' := 'call'}
PROPERTY TrackId : UDINT
GET
TrackId := _TrackId;
END_GET
SET
_TrackId := TrackId;
END_SET
END_PROPERTY

{attribute 'monitoring':='call'}
PROPERTY XtsMoverVisitee : I_AcceptXtsMoverVisitors
GET
XtsMoverVisitee := _Visitee;
END_GET
SET
_Visitee := XtsMoverVisitee;
END_SET
END_PROPERTY

{attribute 'monitoring' := 'call'}
PROPERTY Aborted : BOOL
GET
Aborted := FALSE;
END_GET
END_PROPERTY

{attribute 'monitoring':='call'}
PROPERTY Busy : BOOL
GET
VAR
	Status : I_XtsMoverTaskResult;
END_VAR
_Status.ResetIterator();
WHILE _Status.MoveToNext DO
	__QUERYINTERFACE(_Status.Current, Status);
	IF Status.Busy THEN
		Busy := TRUE;
		RETURN;
	END_IF
END_WHILE
END_GET
END_PROPERTY

PROPERTY CommandExecuted : BOOL
GET
VAR
	Status : I_XtsMoverTaskResult;
END_VAR
_Status.ResetIterator();
WHILE _Status.MoveToNext DO
	__QUERYINTERFACE(_Status.Current, Status);
	IF Status.CommandExecuted THEN
		CommandExecuted := TRUE;
		RETURN;
	END_IF
END_WHILE
END_GET
END_PROPERTY

{attribute 'monitoring':='call'}
PROPERTY Error : BOOL
GET
VAR
	Status : I_XtsMoverTaskResult;
END_VAR
_Status.ResetIterator();
WHILE _Status.MoveToNext DO
	__QUERYINTERFACE(_Status.Current, Status);
	IF Status.Error THEN
		Error := TRUE;
		RETURN;
	END_IF
END_WHILE
END_GET
END_PROPERTY

{attribute 'monitoring':='call'}
PROPERTY ErrorId : UDINT
GET
VAR
	Status : I_XtsMoverTaskResult;
END_VAR
_Status.ResetIterator();
WHILE _Status.MoveToNext DO
	__QUERYINTERFACE(_Status.Current, Status);
	IF Status.Error THEN
		ErrorId := Status.ErrorId;
		RETURN;
	END_IF
END_WHILE
END_GET
END_PROPERTY

METHOD ExecuteOn : I_XtsMoverTaskResult
VAR_INPUT
	Visitee : I_AcceptXtsMoverVisitors;
END_VAR
_Status.Clear();
_Visitee := Visitee;
_Visitee.AcceptMoverVisitor(THIS^);
ExecuteOn := THIS^;
END_METHOD

{attribute 'monitoring' := 'call'}
PROPERTY TaskId : MoverTaskId
GET
TaskId := MoverTaskId.ACTIVATE_TRACK;
END_GET
END_PROPERTY

{attribute 'monitoring' := 'call'}
PROPERTY TaskName : STRING
GET
TaskName := 'Activate Track';
END_GET
END_PROPERTY

METHOD VisitMover
VAR_INPUT
	Mover	: I_XtsMover;
END_VAR
VAR
	Result : I_XtsMoverTaskResult;
END_VAR
Result := Mover.ActivateTrack(_TrackId);
_Status.AddItem(Result);
END_METHOD

END_FUNCTION_BLOCK

// MoverVisitors/XtsMoverHalt
FUNCTION_BLOCK XtsMoverHalt IMPLEMENTS I_XtsMoverVisitor, I_XtsMoverTaskResult, I_CollisionAvoidanceDynamics, I_XtsMoverVisitorTask
VAR
	_Status		  : Collection<XtsCoreParameters.MaxNumberOfMovers>;
	_Visitee	  : I_AcceptXtsMoverVisitors;
	_Deceleration : LREAL;
	_Jerk		  : LREAL;
	_Gap		  : CollisionAvoidanceDynamics;
END_VAR

METHOD CopyParametersFrom
VAR_INPUT
	CopyFrom : I_XtsParameterSet;
END_VAR
_Deceleration := CopyFrom.Deceleration;
_Jerk		  := CopyFrom.Jerk;
_Gap.Gap	  := CopyFrom.Gap;
END_METHOD

{attribute 'monitoring' := 'call'}
PROPERTY Deceleration : LREAL
GET
Deceleration := _Deceleration;
END_GET
SET
_Deceleration := Deceleration;
END_SET
END_PROPERTY

{attribute 'monitoring' := 'call'}
PROPERTY Gap : LREAL
GET
Gap := _Gap.Gap;
END_GET
SET
_Gap.Gap := Gap;
END_SET
END_PROPERTY

{attribute 'monitoring' := 'call'}
PROPERTY Jerk : LREAL
GET
Jerk := _Jerk;
END_GET
SET
_Jerk := Jerk;
END_SET
END_PROPERTY

{attribute 'monitoring':='call'}
PROPERTY XtsMoverVisitee : I_AcceptXtsMoverVisitors
GET
XtsMoverVisitee := _Visitee;
END_GET
SET
_Visitee := XtsMoverVisitee;
END_SET
END_PROPERTY

{attribute 'monitoring' := 'call'}
PROPERTY Aborted : BOOL
GET
END_GET
END_PROPERTY

{attribute 'monitoring':='call'}
PROPERTY Busy : BOOL
GET
VAR
	Status : I_XtsMoverTaskResult;
END_VAR
_Status.ResetIterator();
WHILE _Status.MoveToNext DO
	__QUERYINTERFACE(_Status.Current, Status);
	IF Status.Busy THEN
		Busy := TRUE;
		RETURN;
	END_IF
END_WHILE
END_GET
END_PROPERTY

PROPERTY CommandExecuted : BOOL
GET
VAR
	Status : I_XtsMoverTaskResult;
END_VAR
_Status.ResetIterator();
WHILE _Status.MoveToNext DO
	__QUERYINTERFACE(_Status.Current, Status);
	IF Status.CommandExecuted THEN
		CommandExecuted := TRUE;
		RETURN;
	END_IF
END_WHILE
END_GET
END_PROPERTY

{attribute 'monitoring':='call'}
PROPERTY Error : BOOL
GET
VAR
	Status : I_XtsMoverTaskResult;
END_VAR
_Status.ResetIterator();
WHILE _Status.MoveToNext DO
	__QUERYINTERFACE(_Status.Current, Status);
	IF Status.Error THEN
		Error := TRUE;
		RETURN;
	END_IF
END_WHILE
END_GET
END_PROPERTY

{attribute 'monitoring':='call'}
PROPERTY ErrorId : UDINT
GET
VAR
	Status : I_XtsMoverTaskResult;
END_VAR
_Status.ResetIterator();
WHILE _Status.MoveToNext DO
	__QUERYINTERFACE(_Status.Current, Status);
	IF Status.Error THEN
		ErrorId := Status.ErrorId;
		RETURN;
	END_IF
END_WHILE
END_GET
END_PROPERTY

METHOD ExecuteOn : I_XtsMoverTaskResult
VAR_INPUT
	Visitee  : I_AcceptXtsMoverVisitors;
END_VAR
_Status.Clear();
_Visitee := Visitee;
_Visitee.AcceptMoverVisitor(THIS^);
ExecuteOn := THIS^;
END_METHOD

{attribute 'monitoring' := 'call'}
PROPERTY TaskId : MoverTaskId
GET
TaskId := MoverTaskId.HALT_MOVER;
END_GET
END_PROPERTY

{attribute 'monitoring' := 'call'}
PROPERTY TaskName : STRING
GET
TaskName := 'Halt Mover';
END_GET
END_PROPERTY

METHOD VisitMover
VAR_INPUT
	Mover	: I_XtsMover;
END_VAR
VAR
	Result : I_XtsMoverTaskResult;
END_VAR
Mover.Parameters.Jerk := _Jerk;
Result				  := Mover.Halt(_Deceleration, _Gap.Gap);
_Status.AddItem(Result);
END_METHOD

END_FUNCTION_BLOCK

// MoverVisitors/XtsMoverAddToGroup
FUNCTION_BLOCK XtsMoverAddToGroup IMPLEMENTS I_XtsMoverVisitor, I_XtsMoverTaskResult, I_XtsMoverVisitorTask
VAR
	_Status		  : Collection<XtsCoreParameters.MaxNumberOfMovers>;
	_Visitee	  : I_AcceptXtsMoverVisitors;
	_IdentInGroup : UDINT;
	_AxesGroup	  : REFERENCE TO AXES_GROUP_REF;
END_VAR

{attribute 'monitoring' := 'call'}
PROPERTY AxesGroup : REFERENCE TO AXES_GROUP_REF
GET
AxesGroup REF= _AxesGroup;
END_GET
SET
_AxesGroup REF= AxesGroup;
END_SET
END_PROPERTY

{attribute 'monitoring' := 'call'}
PROPERTY IdentInGroup : UDINT
GET
IdentInGroup := _IdentInGroup;
END_GET
SET
_IdentInGroup := IdentInGroup;
END_SET
END_PROPERTY

{attribute 'monitoring':='call'}
PROPERTY XtsMoverVisitee : I_AcceptXtsMoverVisitors
GET
XtsMoverVisitee := _Visitee;
END_GET
SET
_Visitee := XtsMoverVisitee;
END_SET
END_PROPERTY

{attribute 'monitoring' := 'call'}
PROPERTY Aborted : BOOL
GET
Aborted := FALSE;
END_GET
END_PROPERTY

{attribute 'monitoring':='call'}
PROPERTY Busy : BOOL
GET
VAR
	Status : I_XtsMoverTaskResult;
END_VAR
_Status.ResetIterator();
WHILE _Status.MoveToNext DO
	__QUERYINTERFACE(_Status.Current, Status);
	IF Status.Busy THEN
		Busy := TRUE;
		RETURN;
	END_IF
END_WHILE
END_GET
END_PROPERTY

PROPERTY CommandExecuted : BOOL
GET
VAR
	Status : I_XtsMoverTaskResult;
END_VAR
_Status.ResetIterator();
WHILE _Status.MoveToNext DO
	__QUERYINTERFACE(_Status.Current, Status);
	IF Status.CommandExecuted THEN
		CommandExecuted := TRUE;
		RETURN;
	END_IF
END_WHILE
END_GET
END_PROPERTY

{attribute 'monitoring':='call'}
PROPERTY Error : BOOL
GET
VAR
	Status : I_XtsMoverTaskResult;
END_VAR
_Status.ResetIterator();
WHILE _Status.MoveToNext DO
	__QUERYINTERFACE(_Status.Current, Status);
	IF Status.Error THEN
		Error := TRUE;
		RETURN;
	END_IF
END_WHILE
END_GET
END_PROPERTY

{attribute 'monitoring':='call'}
PROPERTY ErrorId : UDINT
GET
VAR
	Status : I_XtsMoverTaskResult;
END_VAR
_Status.ResetIterator();
WHILE _Status.MoveToNext DO
	__QUERYINTERFACE(_Status.Current, Status);
	IF Status.Error THEN
		ErrorId := Status.ErrorId;
		RETURN;
	END_IF
END_WHILE
END_GET
END_PROPERTY

METHOD ExecuteOn : I_XtsMoverTaskResult
VAR_INPUT
	Visitee : I_AcceptXtsMoverVisitors;
END_VAR
IF NOT __ISVALIDREF(_AxesGroup) THEN
	RETURN;
END_IF

_Status.Clear();
_Visitee := Visitee;
_Visitee.AcceptMoverVisitor(THIS^);
ExecuteOn := THIS^;
END_METHOD

{attribute 'monitoring' := 'call'}
PROPERTY TaskId : MoverTaskId
GET
TaskId := MoverTaskId.ADD_TO_GROUP;
END_GET
END_PROPERTY

{attribute 'monitoring' := 'call'}
PROPERTY TaskName : STRING
GET
TaskName := 'Add Mover To Group';
END_GET
END_PROPERTY

METHOD VisitMover
VAR_INPUT
	Mover	: I_XtsMover;
END_VAR
VAR
	Result : I_XtsMoverTaskResult;
END_VAR
IF Mover.ManualGroupControl THEN
	RETURN;
END_IF

Result		  := Mover.AddToGroup(Group := _AxesGroup, Ident := _IdentInGroup);
_IdentInGroup := _IdentInGroup + 1;
_Status.AddItem(Result);
END_METHOD

END_FUNCTION_BLOCK

// MoverVisitors/XtsMoverRemoveFromGroup
FUNCTION_BLOCK XtsMoverRemoveFromGroup IMPLEMENTS I_XtsMoverVisitor, I_XtsMoverTaskResult, I_XtsMoverVisitorTask
VAR
	_Status		  : Collection<XtsCoreParameters.MaxNumberOfMovers>;
	_Visitee	  : I_AcceptXtsMoverVisitors;
	_IdentInGroup : UDINT;
	_AxesGroup	  : REFERENCE TO AXES_GROUP_REF;
END_VAR

{attribute 'monitoring' := 'call'}
PROPERTY AxesGroup : REFERENCE TO AXES_GROUP_REF
GET
AxesGroup REF= _AxesGroup;
END_GET
SET
_AxesGroup REF= AxesGroup;
END_SET
END_PROPERTY

{attribute 'monitoring' := 'call'}
PROPERTY IdentInGroup : UDINT
GET
IdentInGroup := _IdentInGroup;
END_GET
SET
_IdentInGroup := IdentInGroup;
END_SET
END_PROPERTY

{attribute 'monitoring':='call'}
PROPERTY XtsMoverVisitee : I_AcceptXtsMoverVisitors
GET
XtsMoverVisitee := _Visitee;
END_GET
SET
_Visitee := XtsMoverVisitee;
END_SET
END_PROPERTY

{attribute 'monitoring' := 'call'}
PROPERTY Aborted : BOOL
GET
Aborted := FALSE;
END_GET
END_PROPERTY

{attribute 'monitoring':='call'}
PROPERTY Busy : BOOL
GET
VAR
	Status : I_XtsMoverTaskResult;
END_VAR
_Status.ResetIterator();
WHILE _Status.MoveToNext DO
	__QUERYINTERFACE(_Status.Current, Status);
	IF Status.Busy THEN
		Busy := TRUE;
		RETURN;
	END_IF
END_WHILE
END_GET
END_PROPERTY

PROPERTY CommandExecuted : BOOL
GET
VAR
	Status : I_XtsMoverTaskResult;
END_VAR
_Status.ResetIterator();
WHILE _Status.MoveToNext DO
	__QUERYINTERFACE(_Status.Current, Status);
	IF Status.CommandExecuted THEN
		CommandExecuted := TRUE;
		RETURN;
	END_IF
END_WHILE
END_GET
END_PROPERTY

{attribute 'monitoring':='call'}
PROPERTY Error : BOOL
GET
VAR
	Status : I_XtsMoverTaskResult;
END_VAR
_Status.ResetIterator();
WHILE _Status.MoveToNext DO
	__QUERYINTERFACE(_Status.Current, Status);
	IF Status.Error THEN
		Error := TRUE;
		RETURN;
	END_IF
END_WHILE
END_GET
END_PROPERTY

{attribute 'monitoring':='call'}
PROPERTY ErrorId : UDINT
GET
VAR
	Status : I_XtsMoverTaskResult;
END_VAR
_Status.ResetIterator();
WHILE _Status.MoveToNext DO
	__QUERYINTERFACE(_Status.Current, Status);
	IF Status.Error THEN
		ErrorId := Status.ErrorId;
		RETURN;
	END_IF
END_WHILE
END_GET
END_PROPERTY

METHOD ExecuteOn : I_XtsMoverTaskResult
VAR_INPUT
	Visitee : I_AcceptXtsMoverVisitors;
END_VAR
IF NOT __ISVALIDREF(_AxesGroup) THEN
	RETURN;
END_IF

_Status.Clear();
_Visitee := Visitee;
_Visitee.AcceptMoverVisitor(THIS^);
ExecuteOn := THIS^;
END_METHOD

{attribute 'monitoring' := 'call'}
PROPERTY TaskId : MoverTaskId
GET
TaskId := MoverTaskId.REMOVE_FROM_GROUP;
END_GET
END_PROPERTY

{attribute 'monitoring' := 'call'}
PROPERTY TaskName : STRING
GET
TaskName := 'Remove Mover From Group';
END_GET
END_PROPERTY

METHOD VisitMover
VAR_INPUT
	Mover	: I_XtsMover;
END_VAR
VAR
	Result : I_XtsMoverTaskResult;
END_VAR
IF Mover.ManualGroupControl THEN
	RETURN;
END_IF

Result		  := Mover.RemoveFromGroup(Group := _AxesGroup, Ident := _IdentInGroup);
_IdentInGroup := _IdentInGroup + 1;
_Status.AddItem(Result);
END_METHOD

END_FUNCTION_BLOCK

// _Internal/Mover/Parameters/XtsParameterSet
{attribute 'no_explicit_call' := 'This FB is a CLASS and must be accessed using methods or properties'}
{attribute 'hide_all_locals'}
FUNCTION_BLOCK XtsParameterSet IMPLEMENTS I_XtsParameterSet
VAR
	_CollisionAvoidanceDynamics : CollisionAvoidanceDynamics;
	_BaseDynamics				: BaseDynamics;
	_MoveToPosition				: MoveToPositionParameters;
	_MoveToStation				: MoveToStationParameters;
	_Track						: XtsTrackParameter;
	_SyncAxisParameters			: SyncAxisParameters;
END_VAR

{attribute 'monitoring' := 'call'}
PROPERTY Acceleration : LREAL
GET
Acceleration := _BaseDynamics.Acceleration;
END_GET
SET
_BaseDynamics.Acceleration := Acceleration;
END_SET
END_PROPERTY

METHOD CopyFrom
VAR_INPUT
	Other : I_XtsParameterSet;
END_VAR
Acceleration := Other.Acceleration;
Deceleration := Other.Deceleration;
Velocity	 := Other.Velocity;
Jerk		 := Other.Jerk;
Direction	 := Other.Direction;
Gap			 := Other.Gap;
END_METHOD

METHOD CopyTo
VAR_INPUT
	Other : I_XtsParameterSet;
END_VAR
Other.Acceleration := Acceleration;
Other.Deceleration := Deceleration;
Other.Velocity	   := Velocity;
Other.Jerk		   := Jerk;
Other.Direction	   := Direction;
Other.Gap		   := Gap;
END_METHOD

{attribute 'monitoring' := 'call'}
PROPERTY Deceleration : LREAL
GET
Deceleration := _BaseDynamics.Deceleration;
END_GET
SET
_BaseDynamics.Deceleration := Deceleration;
END_SET
END_PROPERTY

{attribute 'monitoring' := 'call'}
PROPERTY Direction :  Tc3_Mc3Definitions.MC_DIRECTION
GET
Direction := _BaseDynamics.Direction;
END_GET
SET
_BaseDynamics.Direction := Direction;
END_SET
END_PROPERTY

{attribute 'monitoring' := 'call'}
PROPERTY Gap : LREAL
GET
Gap := _CollisionAvoidanceDynamics.Gap;
END_GET
SET
_CollisionAvoidanceDynamics.Gap := Gap;
END_SET
END_PROPERTY

{attribute 'monitoring' := 'call'}
PROPERTY Jerk : LREAL
GET
Jerk := _BaseDynamics.Jerk;
END_GET
SET
_BaseDynamics.Jerk := Jerk;
END_SET
END_PROPERTY

{attribute 'monitoring' := 'call'}
PROPERTY Position : LREAL
GET
Position := _MoveToPosition.Position;
END_GET
SET
_MoveToPosition.Position := Position;
END_SET
END_PROPERTY

{attribute 'monitoring':='call'}
PROPERTY SyncAxis : I_SyncAxisParameters
GET
SyncAxis := _SyncAxisParameters;
END_GET
END_PROPERTY

{attribute 'monitoring' := 'call'}
PROPERTY Track : I_XtsTrack
GET
Track := _Track.Track;
END_GET
SET
_Track.Track := Track;
END_SET
END_PROPERTY

{attribute 'monitoring' := 'call'}
PROPERTY Velocity : LREAL
GET
Velocity := _BaseDynamics.Velocity;
END_GET
SET
_BaseDynamics.Velocity := Velocity;
END_SET
END_PROPERTY

END_FUNCTION_BLOCK

// _Internal/Mover/Parameters/XtsTrackParameter
{attribute 'no_explicit_call' := 'This FB is a CLASS and must be accessed using methods or properties'}
FUNCTION_BLOCK XtsTrackParameter IMPLEMENTS I_XtsTrackParameter
VAR
	_CurrentTrack : I_XtsTrack := NullObjects.XtsTrack;
END_VAR

{attribute 'monitoring' := 'call'}
PROPERTY Track : I_XtsTrack
GET
Track := _CurrentTrack;
END_GET
SET
_CurrentTrack := Track;
END_SET
END_PROPERTY

END_FUNCTION_BLOCK

// _Internal/Tracks/XtsTrack
{attribute 'no_explicit_call' := 'This FB is a CLASS and must be accessed using methods or properties'}
{attribute 'enable_dynamic_creation'}
{attribute 'hide_all_locals'}
FUNCTION_BLOCK XtsTrack IMPLEMENTS I_XtsTrack
VAR
	_Otcid	  : OTCID;
	_Id		  : UDINT;
	_Length	  : LREAL;
	_Offset	  : LREAL;
	_Polarity : Polarity;
	_Utility  : I_TcIoXtsXpuTrack;
END_VAR

METHOD Dispose
VAR
	pDispose : POINTER TO XtsTrack;
END_VAR
pDispose := THIS;
__DELETE(pDispose);
END_METHOD

{attribute 'monitoring' := 'call'}
PROPERTY Id : UDINT
GET
Id := _Id;
END_GET
SET
_Id := Id;
END_SET
END_PROPERTY

{attribute 'monitoring' := 'call'}
PROPERTY Length : LREAL
GET
Length := _Length;
END_GET
SET
_Length := Length;
END_SET
END_PROPERTY

{attribute 'monitoring' := 'call'}
PROPERTY Offset : LREAL
GET
Offset := _Offset;
END_GET
SET
_Offset := Offset;
END_SET
END_PROPERTY

{attribute 'monitoring':='call'}
PROPERTY Otcid : OTCID
GET
Otcid := _Otcid;
END_GET
SET
_Otcid := Otcid;
END_SET
END_PROPERTY

{attribute 'monitoring' := 'call'}
PROPERTY Polarity : Polarity
GET
Polarity := _Polarity;
END_GET
SET
_Polarity := Polarity;
END_SET
END_PROPERTY

PROPERTY Utility : I_TcIoXtsXpuTrack
GET
Utility := _Utility;
END_GET
SET
_Utility := Utility;
END_SET
END_PROPERTY

END_FUNCTION_BLOCK

// _Internal/Mover/Parameters/SyncAxisParameters
{attribute 'no_explicit_call' := 'This FB is a CLASS and must be accessed using methods or properties'}
{attribute 'hide_all_locals'}
FUNCTION_BLOCK SyncAxisParameters IMPLEMENTS I_SyncAxisParameters
VAR
	_MasterAxis			 : REFERENCE TO AXIS_REF;
	_MasterStartDistance : MC_LREAL;
	_MasterSyncPosition	 : MC_LREAL;
	_Options_CA			 : Tc3_McCollisionAvoidance.ST_GearInPosCAOptions;
	_RatioDenominator	 : UINT		:= 1;
	_RatioNumerator		 : MC_LREAL := 1;
	_SlaveSyncPosition	 : MC_LREAL;
	_SyncMode			 : Tc3_McCollisionAvoidance.MC_SYNC_MODE	 := Tc3_McCollisionAvoidance.mcSyncModeNonModulo;
	_SyncStrategy		 : Tc3_McCollisionAvoidance.MC_SYNC_STRATEGY := Tc3_McCollisionAvoidance.mcSyncStrategyEarly;
END_VAR

{attribute 'monitoring':='call'}
PROPERTY MasterAxis : REFERENCE TO AXIS_REF
GET
MasterAxis REF= _MasterAxis;
END_GET
SET
_MasterAxis REF= MasterAxis;
END_SET
END_PROPERTY

{attribute 'monitoring' := 'call'}
PROPERTY MasterStartDistance : MC_LREAL
GET
MasterStartDistance := _MasterStartDistance;
END_GET
SET
END_SET
END_PROPERTY

{attribute 'monitoring' := 'call'}
PROPERTY MasterSyncPosition : MC_LREAL
GET
MasterSyncPosition := _MasterSyncPosition;
END_GET
SET
_MasterSyncPosition := MasterSyncPosition;
END_SET
END_PROPERTY

PROPERTY Options_CA : REFERENCE TO Tc3_McCollisionAvoidance.ST_GearInPosCAOptions
GET
Options_CA REF= _Options_CA;
END_GET
SET
_Options_CA := Options_CA;
END_SET
END_PROPERTY

{attribute 'monitoring' := 'call'}
PROPERTY RatioDenominator : UINT
GET
RatioDenominator := _RatioDenominator;
END_GET
SET
_RatioDenominator := RatioDenominator;
END_SET
END_PROPERTY

{attribute 'monitoring' := 'call'}
PROPERTY RatioNumerator : MC_LREAL
GET
RatioNumerator := _RatioNumerator;
END_GET
SET
_RatioNumerator := RatioNumerator;
END_SET
END_PROPERTY

{attribute 'monitoring' := 'call'}
PROPERTY SlaveSyncPosition : LREAL
GET
SlaveSyncPosition := _SlaveSyncPosition;
END_GET
SET
_SlaveSyncPosition := SlaveSyncPosition;
END_SET
END_PROPERTY

{attribute 'monitoring' := 'call'}
PROPERTY SyncMode : Tc3_McCollisionAvoidance.MC_SYNC_MODE
GET
SyncMode := _SyncMode;
END_GET
SET
_SyncMode := SyncMode;
END_SET
END_PROPERTY

{attribute 'monitoring' := 'call'}
PROPERTY SyncStrategy : Tc3_McCollisionAvoidance.MC_SYNC_STRATEGY
GET
SyncStrategy := _SyncStrategy;
END_GET
SET
_SyncStrategy := SyncStrategy;
END_SET
END_PROPERTY

END_FUNCTION_BLOCK

// _Internal/GroupController/Interfaces/I_ContainXtsMoverGroupController
INTERFACE I_ContainXtsMoverGroupController EXTENDS I_Base

PROPERTY XtsMoverGroupController : I_XtsMoverGroupController
SET
END_SET
END_PROPERTY

END_INTERFACE

// _Internal/GroupController/Interfaces/I_XtsMoverGroupController
INTERFACE I_XtsMoverGroupController EXTENDS I_Base, I_TaskResult, I_Resettable, I_Enablable

{attribute 'monitoring' := 'call'}
PROPERTY AxesGroup : REFERENCE TO AXES_GROUP_REF
SET
END_SET
END_PROPERTY

{attribute 'monitoring':='call'}
PROPERTY GroupStatus : E_MoverGroupState
GET
END_GET
END_PROPERTY

END_INTERFACE

// _Internal/XtsSystem/Tasks/Interfaces/I_XtsMoverIdentificationTask
INTERFACE I_XtsMoverIdentificationTask EXTENDS I_XtsTask, I_Cyclic, I_XtsExecutableTask, I_Resettable

END_INTERFACE

